   S700_BT_CODE_2101.TEST_TEMP[3] := B#16#0;
   S700_BT_CODE_2101.TEST_TEMP[4] := B#16#0;
   S700_BT_CODE_2101.TEST_TEMP[5] := B#16#0;
   S700_BT_CODE_2101.TEST_TEMP[6] := B#16#0;
   S700_BT_CODE_2101.TEST_TEMP[7] := B#16#0;
   S700_BT_CODE_2101.TEST_TEMP[8] := B#16#0;
   S700_BT_CODE_2101.TEST_TEMP[9] := B#16#0;
   S700_BT_CODE_2101.TEST_TEMP[10] := B#16#0;
   S700_BT_CODE_2101.TEST_TEMP[11] := B#16#0;
   S700_BT_CODE_2101.TEST_TEMP[12] := B#16#0;
   S700_BT_CODE_2101.TEST_TEMP[13] := B#16#0;
   S700_BT_CODE_2101.TEST_TEMP[14] := B#16#0;
   S700_BT_CODE_2101.TEST_TEMP[15] := B#16#0;
   S700_BT_CODE_2101.TEST_TEMP[16] := B#16#0;
   S700_BT_CODE_2101.TEST_TEMP[17] := B#16#0;
   S700_BT_CODE_2101.TEST_TEMP[18] := B#16#0;
   S700_BT_CODE_2101.TEST_TEMP[19] := B#16#0;
   S700_BT_CODE_2101.TEST_TEMP[20] := B#16#0;
   S700_BT_CODE_2101.TEST_TEMP[21] := B#16#0;
   S700_BT_CODE_2101.TEST_TEMP[22] := B#16#0;
   S700_BT_CODE_2101.TEST_TEMP[23] := B#16#0;
   S700_BT_CODE_2101.TEST_TEMP[24] := B#16#0;
   S700_BT_CODE_2101.TEST_TEMP[25] := B#16#0;
   S700_BT_CODE_2101.TEST_TEMP[26] := B#16#0;
   S700_BT_CODE_2101.TEST_TEMP[27] := B#16#0;
   S700_BT_CODE_2101.TEST_TEMP[28] := B#16#0;
   S700_BT_CODE_2101.TEST_TEMP[29] := B#16#0;
   S700_BT_CODE_2101.TEST_TEMP[30] := B#16#0;
   S700_BT_CODE_2101.TEST_TEMP[31] := B#16#0;
   S700_BT_CODE_2101.TEST_TEMP[32] := B#16#0;
   S700_BT_CODE_2101.TEST_TEMP[33] := B#16#0;
   S700_BT_CODE_2101.TEST_TEMP[34] := B#16#0;
   S700_BT_CODE_2101.TEST_TEMP[35] := B#16#0;
   S700_BT_CODE_2101.TEST_TEMP[36] := B#16#0;
   S700_BT_CODE_2101.TEST_TEMP[37] := B#16#0;
   S700_BT_CODE_2101.TEST_TEMP[38] := B#16#0;
   S700_BT_CODE_2101.TEST_TEMP[39] := B#16#0;
   S700_BT_CODE_2101.TEST_TEMP[40] := B#16#0;
   S700_BT_CODE_2102.STATION_MAIN := W#16#0;
   S700_BT_CODE_2102.DISTINCTION_LH_RH := W#16#0;
   S700_BT_CODE_2102.STAION_NUMBER := W#16#0;
   S700_BT_CODE_2102.BODY_TYPE_1ST := W#16#0;
   S700_BT_CODE_2102.BODY_TYPE_OPTION := W#16#0;
   S700_BT_CODE_2102.RBT1_STANDARD_WELD_DATA := W#16#0;
   S700_BT_CODE_2102.RBT2_STANDARD_WELD_DATA := W#16#0;
   S700_BT_CODE_2102.RBT3_STANDARD_WELD_DATA := W#16#0;
   S700_BT_CODE_2102.RBT4_STANDARD_WELD_DATA := W#16#0;
   S700_BT_CODE_2102.RBT5_STANDARD_WELD_DATA := W#16#0;
   S700_BT_CODE_2102.RBT6_STANDARD_WELD_DATA := W#16#0;
   S700_BT_CODE_2102.RBT7_STANDARD_WELD_DATA := W#16#0;
   S700_BT_CODE_2102.RBT8_STANDARD_WELD_DATA := W#16#0;
   S700_BT_CODE_2102.RBT9_STANDARD_WELD_DATA := W#16#0;
   S700_BT_CODE_2102.RBT10_STANDARD_WELD_DATA := W#16#0;
   S700_BT_CODE_2102.RBT11_STANDARD_WELD_DATA := W#16#0;
   S700_BT_CODE_2102.RBT12_STANDARD_WELD_DATA := W#16#0;
   S700_BT_CODE_2102.RBT13_STANDARD_WELD_DATA := W#16#0;
   S700_BT_CODE_2102.RBT14_STANDARD_WELD_DATA := W#16#0;
   S700_BT_CODE_2102.RBT15_STANDARD_WELD_DATA := W#16#0;
   S700_BT_CODE_2102.RBT16_STANDARD_WELD_DATA := W#16#0;
   S700_BT_CODE_2102.RBT17_STANDARD_WELD_DATA := W#16#0;
   S700_BT_CODE_2102.RBT18_STANDARD_WELD_DATA := W#16#0;
   S700_BT_CODE_2102.RBT19_STANDARD_WELD_DATA := W#16#0;
   S700_BT_CODE_2102.RBT20_STANDARD_WELD_DATA := W#16#0;
   S700_BT_CODE_2102.RBT21_STANDARD_WELD_DATA := W#16#0;
   S700_BT_CODE_2102.RBT22_STANDARD_WELD_DATA := W#16#0;
   S700_BT_CODE_2102.RBT23_STANDARD_WELD_DAT := W#16#0;
   S700_BT_CODE_2102.RBT24_STANDARD_WELD_DAT := W#16#0;
   S700_BT_CODE_2102.CHK_WORD := W#16#0;
   S700_BT_CODE_2102.TEST_TEMP[1] := B#16#0;
   S700_BT_CODE_2102.TEST_TEMP[2] := B#16#0;
   S700_BT_CODE_2102.TEST_TEMP[3] := B#16#0;
   S700_BT_CODE_2102.TEST_TEMP[4] := B#16#0;
   S700_BT_CODE_2102.TEST_TEMP[5] := B#16#0;
   S700_BT_CODE_2102.TEST_TEMP[6] := B#16#0;
   S700_BT_CODE_2102.TEST_TEMP[7] := B#16#0;
   S700_BT_CODE_2102.TEST_TEMP[8] := B#16#0;
   S700_BT_CODE_2102.TEST_TEMP[9] := B#16#0;
   S700_BT_CODE_2102.TEST_TEMP[10] := B#16#0;
   S700_BT_CODE_2102.TEST_TEMP[11] := B#16#0;
   S700_BT_CODE_2102.TEST_TEMP[12] := B#16#0;
   S700_BT_CODE_2102.TEST_TEMP[13] := B#16#0;
   S700_BT_CODE_2102.TEST_TEMP[14] := B#16#0;
   S700_BT_CODE_2102.TEST_TEMP[15] := B#16#0;
   S700_BT_CODE_2102.TEST_TEMP[16] := B#16#0;
   S700_BT_CODE_2102.TEST_TEMP[17] := B#16#0;
   S700_BT_CODE_2102.TEST_TEMP[18] := B#16#0;
   S700_BT_CODE_2102.TEST_TEMP[19] := B#16#0;
   S700_BT_CODE_2102.TEST_TEMP[20] := B#16#0;
   S700_BT_CODE_2102.TEST_TEMP[21] := B#16#0;
   S700_BT_CODE_2102.TEST_TEMP[22] := B#16#0;
   S700_BT_CODE_2102.TEST_TEMP[23] := B#16#0;
   S700_BT_CODE_2102.TEST_TEMP[24] := B#16#0;
   S700_BT_CODE_2102.TEST_TEMP[25] := B#16#0;
   S700_BT_CODE_2102.TEST_TEMP[26] := B#16#0;
   S700_BT_CODE_2102.TEST_TEMP[27] := B#16#0;
   S700_BT_CODE_2102.TEST_TEMP[28] := B#16#0;
   S700_BT_CODE_2102.TEST_TEMP[29] := B#16#0;
   S700_BT_CODE_2102.TEST_TEMP[30] := B#16#0;
   S700_BT_CODE_2102.TEST_TEMP[31] := B#16#0;
   S700_BT_CODE_2102.TEST_TEMP[32] := B#16#0;
   S700_BT_CODE_2102.TEST_TEMP[33] := B#16#0;
   S700_BT_CODE_2102.TEST_TEMP[34] := B#16#0;
   S700_BT_CODE_2102.TEST_TEMP[35] := B#16#0;
   S700_BT_CODE_2102.TEST_TEMP[36] := B#16#0;
   S700_BT_CODE_2102.TEST_TEMP[37] := B#16#0;
   S700_BT_CODE_2102.TEST_TEMP[38] := B#16#0;
   S700_BT_CODE_2102.TEST_TEMP[39] := B#16#0;
   S700_BT_CODE_2102.TEST_TEMP[40] := B#16#0;
   S700_BT_CODE_2103.STATION_MAIN := W#16#0;
   S700_BT_CODE_2103.DISTINCTION_LH_RH := W#16#0;
   S700_BT_CODE_2103.STAION_NUMBER := W#16#0;
   S700_BT_CODE_2103.BODY_TYPE_1ST := W#16#0;
   S700_BT_CODE_2103.BODY_TYPE_OPTION := W#16#0;
   S700_BT_CODE_2103.RBT1_STANDARD_WELD_DATA := W#16#0;
   S700_BT_CODE_2103.RBT2_STANDARD_WELD_DATA := W#16#0;
   S700_BT_CODE_2103.RBT3_STANDARD_WELD_DATA := W#16#0;
   S700_BT_CODE_2103.RBT4_STANDARD_WELD_DATA := W#16#0;
   S700_BT_CODE_2103.RBT5_STANDARD_WELD_DATA := W#16#0;
   S700_BT_CODE_2103.RBT6_STANDARD_WELD_DATA := W#16#0;
   S700_BT_CODE_2103.RBT7_STANDARD_WELD_DATA := W#16#0;
   S700_BT_CODE_2103.RBT8_STANDARD_WELD_DATA := W#16#0;
   S700_BT_CODE_2103.RBT9_STANDARD_WELD_DATA := W#16#0;
   S700_BT_CODE_2103.RBT10_STANDARD_WELD_DATA := W#16#0;
   S700_BT_CODE_2103.RBT11_STANDARD_WELD_DATA := W#16#0;
   S700_BT_CODE_2103.RBT12_STANDARD_WELD_DATA := W#16#0;
   S700_BT_CODE_2103.RBT13_STANDARD_WELD_DATA := W#16#0;
   S700_BT_CODE_2103.RBT14_STANDARD_WELD_DATA := W#16#0;
   S700_BT_CODE_2103.RBT15_STANDARD_WELD_DATA := W#16#0;
   S700_BT_CODE_2103.RBT16_STANDARD_WELD_DATA := W#16#0;
   S700_BT_CODE_2103.RBT17_STANDARD_WELD_DATA := W#16#0;
   S700_BT_CODE_2103.RBT18_STANDARD_WELD_DATA := W#16#0;
   S700_BT_CODE_2103.RBT19_STANDARD_WELD_DATA := W#16#0;
   S700_BT_CODE_2103.RBT20_STANDARD_WELD_DATA := W#16#0;
   S700_BT_CODE_2103.RBT21_STANDARD_WELD_DATA := W#16#0;
   S700_BT_CODE_2103.RBT22_STANDARD_WELD_DATA := W#16#0;
   S700_BT_CODE_2103.RBT23_STANDARD_WELD_DAT := W#16#0;
   S700_BT_CODE_2103.RBT24_STANDARD_WELD_DAT := W#16#0;
   S700_BT_CODE_2103.CHK_WORD := W#16#0;
   S700_BT_CODE_2103.TEST_TEMP[1] := B#16#0;
   S700_BT_CODE_2103.TEST_TEMP[2] := B#16#0;
   S700_BT_CODE_2103.TEST_TEMP[3] := B#16#0;
   S700_BT_CODE_2103.TEST_TEMP[4] := B#16#0;
   S700_BT_CODE_2103.TEST_TEMP[5] := B#16#0;
   S700_BT_CODE_2103.TEST_TEMP[6] := B#16#0;
   S700_BT_CODE_2103.TEST_TEMP[7] := B#16#0;
   S700_BT_CODE_2103.TEST_TEMP[8] := B#16#0;
   S700_BT_CODE_2103.TEST_TEMP[9] := B#16#0;
   S700_BT_CODE_2103.TEST_TEMP[10] := B#16#0;
   S700_BT_CODE_2103.TEST_TEMP[11] := B#16#0;
   S700_BT_CODE_2103.TEST_TEMP[12] := B#16#0;
   S700_BT_CODE_2103.TEST_TEMP[13] := B#16#0;
   S700_BT_CODE_2103.TEST_TEMP[14] := B#16#0;
   S700_BT_CODE_2103.TEST_TEMP[15] := B#16#0;
   S700_BT_CODE_2103.TEST_TEMP[16] := B#16#0;
   S700_BT_CODE_2103.TEST_TEMP[17] := B#16#0;
   S700_BT_CODE_2103.TEST_TEMP[18] := B#16#0;
   S700_BT_CODE_2103.TEST_TEMP[19] := B#16#0;
   S700_BT_CODE_2103.TEST_TEMP[20] := B#16#0;
   S700_BT_CODE_2103.TEST_TEMP[21] := B#16#0;
   S700_BT_CODE_2103.TEST_TEMP[22] := B#16#0;
   S700_BT_CODE_2103.TEST_TEMP[23] := B#16#0;
   S700_BT_CODE_2103.TEST_TEMP[24] := B#16#0;
   S700_BT_CODE_2103.TEST_TEMP[25] := B#16#0;
   S700_BT_CODE_2103.TEST_TEMP[26] := B#16#0;
   S700_BT_CODE_2103.TEST_TEMP[27] := B#16#0;
   S700_BT_CODE_2103.TEST_TEMP[28] := B#16#0;
   S700_BT_CODE_2103.TEST_TEMP[29] := B#16#0;
   S700_BT_CODE_2103.TEST_TEMP[30] := B#16#0;
   S700_BT_CODE_2103.TEST_TEMP[31] := B#16#0;
   S700_BT_CODE_2103.TEST_TEMP[32] := B#16#0;
   S700_BT_CODE_2103.TEST_TEMP[33] := B#16#0;
   S700_BT_CODE_2103.TEST_TEMP[34] := B#16#0;
   S700_BT_CODE_2103.TEST_TEMP[35] := B#16#0;
   S700_BT_CODE_2103.TEST_TEMP[36] := B#16#0;
   S700_BT_CODE_2103.TEST_TEMP[37] := B#16#0;
   S700_BT_CODE_2103.TEST_TEMP[38] := B#16#0;
   S700_BT_CODE_2103.TEST_TEMP[39] := B#16#0;
   S700_BT_CODE_2103.TEST_TEMP[40] := B#16#0;
   S700_BT_CODE_2104.STATION_MAIN := W#16#0;
   S700_BT_CODE_2104.DISTINCTION_LH_RH := W#16#0;
   S700_BT_CODE_2104.STAION_NUMBER := W#16#0;
   S700_BT_CODE_2104.BODY_TYPE_1ST := W#16#0;
   S700_BT_CODE_2104.BODY_TYPE_OPTION := W#16#0;
   S700_BT_CODE_2104.RBT1_STANDARD_WELD_DATA := W#16#0;
   S700_BT_CODE_2104.RBT2_STANDARD_WELD_DATA := W#16#0;
   S700_BT_CODE_2104.RBT3_STANDARD_WELD_DATA := W#16#0;
   S700_BT_CODE_2104.RBT4_STANDARD_WELD_DATA := W#16#0;
   S700_BT_CODE_2104.RBT5_STANDARD_WELD_DATA := W#16#0;
   S700_BT_CODE_2104.RBT6_STANDARD_WELD_DATA := W#16#0;
   S700_BT_CODE_2104.RBT7_STANDARD_WELD_DATA := W#16#0;
   S700_BT_CODE_2104.RBT8_STANDARD_WELD_DATA := W#16#0;
   S700_BT_CODE_2104.RBT9_STANDARD_WELD_DATA := W#16#0;
   S700_BT_CODE_2104.RBT10_STANDARD_WELD_DATA := W#16#0;
   S700_BT_CODE_2104.RBT11_STANDARD_WELD_DATA := W#16#0;
   S700_BT_CODE_2104.RBT12_STANDARD_WELD_DATA := W#16#0;
   S700_BT_CODE_2104.RBT13_STANDARD_WELD_DATA := W#16#0;
   S700_BT_CODE_2104.RBT14_STANDARD_WELD_DATA := W#16#0;
   S700_BT_CODE_2104.RBT15_STANDARD_WELD_DATA := W#16#0;
   S700_BT_CODE_2104.RBT16_STANDARD_WELD_DATA := W#16#0;
   S700_BT_CODE_2104.RBT17_STANDARD_WELD_DATA := W#16#0;
   S700_BT_CODE_2104.RBT18_STANDARD_WELD_DATA := W#16#0;
   S700_BT_CODE_2104.RBT19_STANDARD_WELD_DATA := W#16#0;
   S700_BT_CODE_2104.RBT20_STANDARD_WELD_DATA := W#16#0;
   S700_BT_CODE_2104.RBT21_STANDARD_WELD_DATA := W#16#0;
   S700_BT_CODE_2104.RBT22_STANDARD_WELD_DATA := W#16#0;
   S700_BT_CODE_2104.RBT23_STANDARD_WELD_DAT := W#16#0;
   S700_BT_CODE_2104.RBT24_STANDARD_WELD_DAT := W#16#0;
   S700_BT_CODE_2104.CHK_WORD := W#16#0;
   S700_BT_CODE_2104.TEST_TEMP[1] := B#16#0;
   S700_BT_CODE_2104.TEST_TEMP[2] := B#16#0;
   S700_BT_CODE_2104.TEST_TEMP[3] := B#16#0;
   S700_BT_CODE_2104.TEST_TEMP[4] := B#16#0;
   S700_BT_CODE_2104.TEST_TEMP[5] := B#16#0;
   S700_BT_CODE_2104.TEST_TEMP[6] := B#16#0;
   S700_BT_CODE_2104.TEST_TEMP[7] := B#16#0;
   S700_BT_CODE_2104.TEST_TEMP[8] := B#16#0;
   S700_BT_CODE_2104.TEST_TEMP[9] := B#16#0;
   S700_BT_CODE_2104.TEST_TEMP[10] := B#16#0;
   S700_BT_CODE_2104.TEST_TEMP[11] := B#16#0;
   S700_BT_CODE_2104.TEST_TEMP[12] := B#16#0;
   S700_BT_CODE_2104.TEST_TEMP[13] := B#16#0;
   S700_BT_CODE_2104.TEST_TEMP[14] := B#16#0;
   S700_BT_CODE_2104.TEST_TEMP[15] := B#16#0;
   S700_BT_CODE_2104.TEST_TEMP[16] := B#16#0;
   S700_BT_CODE_2104.TEST_TEMP[17] := B#16#0;
   S700_BT_CODE_2104.TEST_TEMP[18] := B#16#0;
   S700_BT_CODE_2104.TEST_TEMP[19] := B#16#0;
   S700_BT_CODE_2104.TEST_TEMP[20] := B#16#0;
   S700_BT_CODE_2104.TEST_TEMP[21] := B#16#0;
   S700_BT_CODE_2104.TEST_TEMP[22] := B#16#0;
   S700_BT_CODE_2104.TEST_TEMP[23] := B#16#0;
   S700_BT_CODE_2104.TEST_TEMP[24] := B#16#0;
   S700_BT_CODE_2104.TEST_TEMP[25] := B#16#0;
   S700_BT_CODE_2104.TEST_TEMP[26] := B#16#0;
   S700_BT_CODE_2104.TEST_TEMP[27] := B#16#0;
   S700_BT_CODE_2104.TEST_TEMP[28] := B#16#0;
   S700_BT_CODE_2104.TEST_TEMP[29] := B#16#0;
   S700_BT_CODE_2104.TEST_TEMP[30] := B#16#0;
   S700_BT_CODE_2104.TEST_TEMP[31] := B#16#0;
   S700_BT_CODE_2104.TEST_TEMP[32] := B#16#0;
   S700_BT_CODE_2104.TEST_TEMP[33] := B#16#0;
   S700_BT_CODE_2104.TEST_TEMP[34] := B#16#0;
   S700_BT_CODE_2104.TEST_TEMP[35] := B#16#0;
   S700_BT_CODE_2104.TEST_TEMP[36] := B#16#0;
   S700_BT_CODE_2104.TEST_TEMP[37] := B#16#0;
   S700_BT_CODE_2104.TEST_TEMP[38] := B#16#0;
   S700_BT_CODE_2104.TEST_TEMP[39] := B#16#0;
   S700_BT_CODE_2104.TEST_TEMP[40] := B#16#0;
   S700_BT_CODE_2105.STATION_MAIN := W#16#0;
   S700_BT_CODE_2105.DISTINCTION_LH_RH := W#16#0;
   S700_BT_CODE_2105.STAION_NUMBER := W#16#0;
   S700_BT_CODE_2105.BODY_TYPE_1ST := W#16#0;
   S700_BT_CODE_2105.BODY_TYPE_OPTION := W#16#0;
   S700_BT_CODE_2105.RBT1_STANDARD_WELD_DATA := W#16#0;
   S700_BT_CODE_2105.RBT2_STANDARD_WELD_DATA := W#16#0;
   S700_BT_CODE_2105.RBT3_STANDARD_WELD_DATA := W#16#0;
   S700_BT_CODE_2105.RBT4_STANDARD_WELD_DATA := W#16#0;
   S700_BT_CODE_2105.RBT5_STANDARD_WELD_DATA := W#16#0;
   S700_BT_CODE_2105.RBT6_STANDARD_WELD_DATA := W#16#0;
   S700_BT_CODE_2105.RBT7_STANDARD_WELD_DATA := W#16#0;
   S700_BT_CODE_2105.RBT8_STANDARD_WELD_DATA := W#16#0;
   S700_BT_CODE_2105.RBT9_STANDARD_WELD_DATA := W#16#0;
   S700_BT_CODE_2105.RBT10_STANDARD_WELD_DATA := W#16#0;
   S700_BT_CODE_2105.RBT11_STANDARD_WELD_DATA := W#16#0;
   S700_BT_CODE_2105.RBT12_STANDARD_WELD_DATA := W#16#0;
   S700_BT_CODE_2105.RBT13_STANDARD_WELD_DATA := W#16#0;
   S700_BT_CODE_2105.RBT14_STANDARD_WELD_DATA := W#16#0;
   S700_BT_CODE_2105.RBT15_STANDARD_WELD_DATA := W#16#0;
   S700_BT_CODE_2105.RBT16_STANDARD_WELD_DATA := W#16#0;
   S700_BT_CODE_2105.RBT17_STANDARD_WELD_DATA := W#16#0;
   S700_BT_CODE_2105.RBT18_STANDARD_WELD_DATA := W#16#0;
   S700_BT_CODE_2105.RBT19_STANDARD_WELD_DATA := W#16#0;
   S700_BT_CODE_2105.RBT20_STANDARD_WELD_DATA := W#16#0;
   S700_BT_CODE_2105.RBT21_STANDARD_WELD_DATA := W#16#0;
   S700_BT_CODE_2105.RBT22_STANDARD_WELD_DATA := W#16#0;
   S700_BT_CODE_2105.RBT23_STANDARD_WELD_DAT := W#16#0;
   S700_BT_CODE_2105.RBT24_STANDARD_WELD_DAT := W#16#0;
   S700_BT_CODE_2105.CHK_WORD := W#16#0;
   S700_BT_CODE_2105.TEST_TEMP[1] := B#16#0;
   S700_BT_CODE_2105.TEST_TEMP[2] := B#16#0;
   S700_BT_CODE_2105.TEST_TEMP[3] := B#16#0;
   S700_BT_CODE_2105.TEST_TEMP[4] := B#16#0;
   S700_BT_CODE_2105.TEST_TEMP[5] := B#16#0;
   S700_BT_CODE_2105.TEST_TEMP[6] := B#16#0;
   S700_BT_CODE_2105.TEST_TEMP[7] := B#16#0;
   S700_BT_CODE_2105.TEST_TEMP[8] := B#16#0;
   S700_BT_CODE_2105.TEST_TEMP[9] := B#16#0;
   S700_BT_CODE_2105.TEST_TEMP[10] := B#16#0;
   S700_BT_CODE_2105.TEST_TEMP[11] := B#16#0;
   S700_BT_CODE_2105.TEST_TEMP[12] := B#16#0;
   S700_BT_CODE_2105.TEST_TEMP[13] := B#16#0;
   S700_BT_CODE_2105.TEST_TEMP[14] := B#16#0;
   S700_BT_CODE_2105.TEST_TEMP[15] := B#16#0;
   S700_BT_CODE_2105.TEST_TEMP[16] := B#16#0;
   S700_BT_CODE_2105.TEST_TEMP[17] := B#16#0;
   S700_BT_CODE_2105.TEST_TEMP[18] := B#16#0;
   S700_BT_CODE_2105.TEST_TEMP[19] := B#16#0;
   S700_BT_CODE_2105.TEST_TEMP[20] := B#16#0;
   S700_BT_CODE_2105.TEST_TEMP[21] := B#16#0;
   S700_BT_CODE_2105.TEST_TEMP[22] := B#16#0;
   S700_BT_CODE_2105.TEST_TEMP[23] := B#16#0;
   S700_BT_CODE_2105.TEST_TEMP[24] := B#16#0;
   S700_BT_CODE_2105.TEST_TEMP[25] := B#16#0;
   S700_BT_CODE_2105.TEST_TEMP[26] := B#16#0;
   S700_BT_CODE_2105.TEST_TEMP[27] := B#16#0;
   S700_BT_CODE_2105.TEST_TEMP[28] := B#16#0;
   S700_BT_CODE_2105.TEST_TEMP[29] := B#16#0;
   S700_BT_CODE_2105.TEST_TEMP[30] := B#16#0;
   S700_BT_CODE_2105.TEST_TEMP[31] := B#16#0;
   S700_BT_CODE_2105.TEST_TEMP[32] := B#16#0;
   S700_BT_CODE_2105.TEST_TEMP[33] := B#16#0;
   S700_BT_CODE_2105.TEST_TEMP[34] := B#16#0;
   S700_BT_CODE_2105.TEST_TEMP[35] := B#16#0;
   S700_BT_CODE_2105.TEST_TEMP[36] := B#16#0;
   S700_BT_CODE_2105.TEST_TEMP[37] := B#16#0;
   S700_BT_CODE_2105.TEST_TEMP[38] := B#16#0;
   S700_BT_CODE_2105.TEST_TEMP[39] := B#16#0;
   S700_BT_CODE_2105.TEST_TEMP[40] := B#16#0;
   S700_BT_CODE_2106.STATION_MAIN := W#16#0;
   S700_BT_CODE_2106.DISTINCTION_LH_RH := W#16#0;
   S700_BT_CODE_2106.STAION_NUMBER := W#16#0;
   S700_BT_CODE_2106.BODY_TYPE_1ST := W#16#0;
   S700_BT_CODE_2106.BODY_TYPE_OPTION := W#16#0;
   S700_BT_CODE_2106.RBT1_STANDARD_WELD_DATA := W#16#0;
   S700_BT_CODE_2106.RBT2_STANDARD_WELD_DATA := W#16#0;
   S700_BT_CODE_2106.RBT3_STANDARD_WELD_DATA := W#16#0;
   S700_BT_CODE_2106.RBT4_STANDARD_WELD_DATA := W#16#0;
   S700_BT_CODE_2106.RBT5_STANDARD_WELD_DATA := W#16#0;
   S700_BT_CODE_2106.RBT6_STANDARD_WELD_DATA := W#16#0;
   S700_BT_CODE_2106.RBT7_STANDARD_WELD_DATA := W#16#0;
   S700_BT_CODE_2106.RBT8_STANDARD_WELD_DATA := W#16#0;
   S700_BT_CODE_2106.RBT9_STANDARD_WELD_DATA := W#16#0;
   S700_BT_CODE_2106.RBT10_STANDARD_WELD_DATA := W#16#0;
   S700_BT_CODE_2106.RBT11_STANDARD_WELD_DATA := W#16#0;
   S700_BT_CODE_2106.RBT12_STANDARD_WELD_DATA := W#16#0;
   S700_BT_CODE_2106.RBT13_STANDARD_WELD_DATA := W#16#0;
   S700_BT_CODE_2106.RBT14_STANDARD_WELD_DATA := W#16#0;
   S700_BT_CODE_2106.RBT15_STANDARD_WELD_DATA := W#16#0;
   S700_BT_CODE_2106.RBT16_STANDARD_WELD_DATA := W#16#0;
   S700_BT_CODE_2106.RBT17_STANDARD_WELD_DATA := W#16#0;
   S700_BT_CODE_2106.RBT18_STANDARD_WELD_DATA := W#16#0;
   S700_BT_CODE_2106.RBT19_STANDARD_WELD_DATA := W#16#0;
   S700_BT_CODE_2106.RBT20_STANDARD_WELD_DATA := W#16#0;
   S700_BT_CODE_2106.RBT21_STANDARD_WELD_DATA := W#16#0;
   S700_BT_CODE_2106.RBT22_STANDARD_WELD_DATA := W#16#0;
   S700_BT_CODE_2106.RBT23_STANDARD_WELD_DAT := W#16#0;
   S700_BT_CODE_2106.RBT24_STANDARD_WELD_DAT := W#16#0;
   S700_BT_CODE_2106.CHK_WORD := W#16#0;
   S700_BT_CODE_2106.TEST_TEMP[1] := B#16#0;
   S700_BT_CODE_2106.TEST_TEMP[2] := B#16#0;
   S700_BT_CODE_2106.TEST_TEMP[3] := B#16#0;
   S700_BT_CODE_2106.TEST_TEMP[4] := B#16#0;
   S700_BT_CODE_2106.TEST_TEMP[5] := B#16#0;
   S700_BT_CODE_2106.TEST_TEMP[6] := B#16#0;
   S700_BT_CODE_2106.TEST_TEMP[7] := B#16#0;
   S700_BT_CODE_2106.TEST_TEMP[8] := B#16#0;
   S700_BT_CODE_2106.TEST_TEMP[9] := B#16#0;
   S700_BT_CODE_2106.TEST_TEMP[10] := B#16#0;
   S700_BT_CODE_2106.TEST_TEMP[11] := B#16#0;
   S700_BT_CODE_2106.TEST_TEMP[12] := B#16#0;
   S700_BT_CODE_2106.TEST_TEMP[13] := B#16#0;
   S700_BT_CODE_2106.TEST_TEMP[14] := B#16#0;
   S700_BT_CODE_2106.TEST_TEMP[15] := B#16#0;
   S700_BT_CODE_2106.TEST_TEMP[16] := B#16#0;
   S700_BT_CODE_2106.TEST_TEMP[17] := B#16#0;
   S700_BT_CODE_2106.TEST_TEMP[18] := B#16#0;
   S700_BT_CODE_2106.TEST_TEMP[19] := B#16#0;
   S700_BT_CODE_2106.TEST_TEMP[20] := B#16#0;
   S700_BT_CODE_2106.TEST_TEMP[21] := B#16#0;
   S700_BT_CODE_2106.TEST_TEMP[22] := B#16#0;
   S700_BT_CODE_2106.TEST_TEMP[23] := B#16#0;
   S700_BT_CODE_2106.TEST_TEMP[24] := B#16#0;
   S700_BT_CODE_2106.TEST_TEMP[25] := B#16#0;
   S700_BT_CODE_2106.TEST_TEMP[26] := B#16#0;
   S700_BT_CODE_2106.TEST_TEMP[27] := B#16#0;
   S700_BT_CODE_2106.TEST_TEMP[28] := B#16#0;
   S700_BT_CODE_2106.TEST_TEMP[29] := B#16#0;
   S700_BT_CODE_2106.TEST_TEMP[30] := B#16#0;
   S700_BT_CODE_2106.TEST_TEMP[31] := B#16#0;
   S700_BT_CODE_2106.TEST_TEMP[32] := B#16#0;
   S700_BT_CODE_2106.TEST_TEMP[33] := B#16#0;
   S700_BT_CODE_2106.TEST_TEMP[34] := B#16#0;
   S700_BT_CODE_2106.TEST_TEMP[35] := B#16#0;
   S700_BT_CODE_2106.TEST_TEMP[36] := B#16#0;
   S700_BT_CODE_2106.TEST_TEMP[37] := B#16#0;
   S700_BT_CODE_2106.TEST_TEMP[38] := B#16#0;
   S700_BT_CODE_2106.TEST_TEMP[39] := B#16#0;
   S700_BT_CODE_2106.TEST_TEMP[40] := B#16#0;
   S700_BT_CODE_2107.STATION_MAIN := W#16#0;
   S700_BT_CODE_2107.DISTINCTION_LH_RH := W#16#0;
   S700_BT_CODE_2107.STAION_NUMBER := W#16#0;
   S700_BT_CODE_2107.BODY_TYPE_1ST := W#16#0;
   S700_BT_CODE_2107.BODY_TYPE_OPTION := W#16#0;
   S700_BT_CODE_2107.RBT1_STANDARD_WELD_DATA := W#16#0;
   S700_BT_CODE_2107.RBT2_STANDARD_WELD_DATA := W#16#0;
   S700_BT_CODE_2107.RBT3_STANDARD_WELD_DATA := W#16#0;
   S700_BT_CODE_2107.RBT4_STANDARD_WELD_DATA := W#16#0;
   S700_BT_CODE_2107.RBT5_STANDARD_WELD_DATA := W#16#0;
   S700_BT_CODE_2107.RBT6_STANDARD_WELD_DATA := W#16#0;
   S700_BT_CODE_2107.RBT7_STANDARD_WELD_DATA := W#16#0;
   S700_BT_CODE_2107.RBT8_STANDARD_WELD_DATA := W#16#0;
   S700_BT_CODE_2107.RBT9_STANDARD_WELD_DATA := W#16#0;
   S700_BT_CODE_2107.RBT10_STANDARD_WELD_DATA := W#16#0;
   S700_BT_CODE_2107.RBT11_STANDARD_WELD_DATA := W#16#0;
   S700_BT_CODE_2107.RBT12_STANDARD_WELD_DATA := W#16#0;
   S700_BT_CODE_2107.RBT13_STANDARD_WELD_DATA := W#16#0;
   S700_BT_CODE_2107.RBT14_STANDARD_WELD_DATA := W#16#0;
   S700_BT_CODE_2107.RBT15_STANDARD_WELD_DATA := W#16#0;
   S700_BT_CODE_2107.RBT16_STANDARD_WELD_DATA := W#16#0;
   S700_BT_CODE_2107.RBT17_STANDARD_WELD_DATA := W#16#0;
   S700_BT_CODE_2107.RBT18_STANDARD_WELD_DATA := W#16#0;
   S700_BT_CODE_2107.RBT19_STANDARD_WELD_DATA := W#16#0;
   S700_BT_CODE_2107.RBT20_STANDARD_WELD_DATA := W#16#0;
   S700_BT_CODE_2107.RBT21_STANDARD_WELD_DATA := W#16#0;
   S700_BT_CODE_2107.RBT22_STANDARD_WELD_DATA := W#16#0;
   S700_BT_CODE_2107.RBT23_STANDARD_WELD_DAT := W#16#0;
   S700_BT_CODE_2107.RBT24_STANDARD_WELD_DAT := W#16#0;
   S700_BT_CODE_2107.CHK_WORD := W#16#0;
   S700_BT_CODE_2107.TEST_TEMP[1] := B#16#0;
   S700_BT_CODE_2107.TEST_TEMP[2] := B#16#0;
   S700_BT_CODE_2107.TEST_TEMP[3] := B#16#0;
   S700_BT_CODE_2107.TEST_TEMP[4] := B#16#0;
   S700_BT_CODE_2107.TEST_TEMP[5] := B#16#0;
   S700_BT_CODE_2107.TEST_TEMP[6] := B#16#0;
   S700_BT_CODE_2107.TEST_TEMP[7] := B#16#0;
   S700_BT_CODE_2107.TEST_TEMP[8] := B#16#0;
   S700_BT_CODE_2107.TEST_TEMP[9] := B#16#0;
   S700_BT_CODE_2107.TEST_TEMP[10] := B#16#0;
   S700_BT_CODE_2107.TEST_TEMP[11] := B#16#0;
   S700_BT_CODE_2107.TEST_TEMP[12] := B#16#0;
   S700_BT_CODE_2107.TEST_TEMP[13] := B#16#0;
   S700_BT_CODE_2107.TEST_TEMP[14] := B#16#0;
   S700_BT_CODE_2107.TEST_TEMP[15] := B#16#0;
   S700_BT_CODE_2107.TEST_TEMP[16] := B#16#0;
   S700_BT_CODE_2107.TEST_TEMP[17] := B#16#0;
   S700_BT_CODE_2107.TEST_TEMP[18] := B#16#0;
   S700_BT_CODE_2107.TEST_TEMP[19] := B#16#0;
   S700_BT_CODE_2107.TEST_TEMP[20] := B#16#0;
   S700_BT_CODE_2107.TEST_TEMP[21] := B#16#0;
   S700_BT_CODE_2107.TEST_TEMP[22] := B#16#0;
   S700_BT_CODE_2107.TEST_TEMP[23] := B#16#0;
   S700_BT_CODE_2107.TEST_TEMP[24] := B#16#0;
   S700_BT_CODE_2107.TEST_TEMP[25] := B#16#0;
   S700_BT_CODE_2107.TEST_TEMP[26] := B#16#0;
   S700_BT_CODE_2107.TEST_TEMP[27] := B#16#0;
   S700_BT_CODE_2107.TEST_TEMP[28] := B#16#0;
   S700_BT_CODE_2107.TEST_TEMP[29] := B#16#0;
   S700_BT_CODE_2107.TEST_TEMP[30] := B#16#0;
   S700_BT_CODE_2107.TEST_TEMP[31] := B#16#0;
   S700_BT_CODE_2107.TEST_TEMP[32] := B#16#0;
   S700_BT_CODE_2107.TEST_TEMP[33] := B#16#0;
   S700_BT_CODE_2107.TEST_TEMP[34] := B#16#0;
   S700_BT_CODE_2107.TEST_TEMP[35] := B#16#0;
   S700_BT_CODE_2107.TEST_TEMP[36] := B#16#0;
   S700_BT_CODE_2107.TEST_TEMP[37] := B#16#0;
   S700_BT_CODE_2107.TEST_TEMP[38] := B#16#0;
   S700_BT_CODE_2107.TEST_TEMP[39] := B#16#0;
   S700_BT_CODE_2107.TEST_TEMP[40] := B#16#0;
   S700_BT_CODE_2108.STATION_MAIN := W#16#0;
   S700_BT_CODE_2108.DISTINCTION_LH_RH := W#16#0;
   S700_BT_CODE_2108.STAION_NUMBER := W#16#0;
   S700_BT_CODE_2108.BODY_TYPE_1ST := W#16#0;
   S700_BT_CODE_2108.BODY_TYPE_OPTION := W#16#0;
   S700_BT_CODE_2108.RBT1_STANDARD_WELD_DATA := W#16#0;
   S700_BT_CODE_2108.RBT2_STANDARD_WELD_DATA := W#16#0;
   S700_BT_CODE_2108.RBT3_STANDARD_WELD_DATA := W#16#0;
   S700_BT_CODE_2108.RBT4_STANDARD_WELD_DATA := W#16#0;
   S700_BT_CODE_2108.RBT5_STANDARD_WELD_DATA := W#16#0;
   S700_BT_CODE_2108.RBT6_STANDARD_WELD_DATA := W#16#0;
   S700_BT_CODE_2108.RBT7_STANDARD_WELD_DATA := W#16#0;
   S700_BT_CODE_2108.RBT8_STANDARD_WELD_DATA := W#16#0;
   S700_BT_CODE_2108.RBT9_STANDARD_WELD_DATA := W#16#0;
   S700_BT_CODE_2108.RBT10_STANDARD_WELD_DATA := W#16#0;
   S700_BT_CODE_2108.RBT11_STANDARD_WELD_DATA := W#16#0;
   S700_BT_CODE_2108.RBT12_STANDARD_WELD_DATA := W#16#0;
   S700_BT_CODE_2108.RBT13_STANDARD_WELD_DATA := W#16#0;
   S700_BT_CODE_2108.RBT14_STANDARD_WELD_DATA := W#16#0;
   S700_BT_CODE_2108.RBT15_STANDARD_WELD_DATA := W#16#0;
   S700_BT_CODE_2108.RBT16_STANDARD_WELD_DATA := W#16#0;
   S700_BT_CODE_2108.RBT17_STANDARD_WELD_DATA := W#16#0;
   S700_BT_CODE_2108.RBT18_STANDARD_WELD_DATA := W#16#0;
   S700_BT_CODE_2108.RBT19_STANDARD_WELD_DATA := W#16#0;
   S700_BT_CODE_2108.RBT20_STANDARD_WELD_DATA := W#16#0;
   S700_BT_CODE_2108.RBT21_STANDARD_WELD_DATA := W#16#0;
   S700_BT_CODE_2108.RBT22_STANDARD_WELD_DATA := W#16#0;
   S700_BT_CODE_2108.RBT23_STANDARD_WELD_DAT := W#16#0;
   S700_BT_CODE_2108.RBT24_STANDARD_WELD_DAT := W#16#0;
   S700_BT_CODE_2108.CHK_WORD := W#16#0;
   S700_BT_CODE_2108.TEST_TEMP[1] := B#16#0;
   S700_BT_CODE_2108.TEST_TEMP[2] := B#16#0;
   S700_BT_CODE_2108.TEST_TEMP[3] := B#16#0;
   S700_BT_CODE_2108.TEST_TEMP[4] := B#16#0;
   S700_BT_CODE_2108.TEST_TEMP[5] := B#16#0;
   S700_BT_CODE_2108.TEST_TEMP[6] := B#16#0;
   S700_BT_CODE_2108.TEST_TEMP[7] := B#16#0;
   S700_BT_CODE_2108.TEST_TEMP[8] := B#16#0;
   S700_BT_CODE_2108.TEST_TEMP[9] := B#16#0;
   S700_BT_CODE_2108.TEST_TEMP[10] := B#16#0;
   S700_BT_CODE_2108.TEST_TEMP[11] := B#16#0;
   S700_BT_CODE_2108.TEST_TEMP[12] := B#16#0;
   S700_BT_CODE_2108.TEST_TEMP[13] := B#16#0;
   S700_BT_CODE_2108.TEST_TEMP[14] := B#16#0;
   S700_BT_CODE_2108.TEST_TEMP[15] := B#16#0;
   S700_BT_CODE_2108.TEST_TEMP[16] := B#16#0;
   S700_BT_CODE_2108.TEST_TEMP[17] := B#16#0;
   S700_BT_CODE_2108.TEST_TEMP[18] := B#16#0;
   S700_BT_CODE_2108.TEST_TEMP[19] := B#16#0;
   S700_BT_CODE_2108.TEST_TEMP[20] := B#16#0;
   S700_BT_CODE_2108.TEST_TEMP[21] := B#16#0;
   S700_BT_CODE_2108.TEST_TEMP[22] := B#16#0;
   S700_BT_CODE_2108.TEST_TEMP[23] := B#16#0;
   S700_BT_CODE_2108.TEST_TEMP[24] := B#16#0;
   S700_BT_CODE_2108.TEST_TEMP[25] := B#16#0;
   S700_BT_CODE_2108.TEST_TEMP[26] := B#16#0;
   S700_BT_CODE_2108.TEST_TEMP[27] := B#16#0;
   S700_BT_CODE_2108.TEST_TEMP[28] := B#16#0;
   S700_BT_CODE_2108.TEST_TEMP[29] := B#16#0;
   S700_BT_CODE_2108.TEST_TEMP[30] := B#16#0;
   S700_BT_CODE_2108.TEST_TEMP[31] := B#16#0;
   S700_BT_CODE_2108.TEST_TEMP[32] := B#16#0;
   S700_BT_CODE_2108.TEST_TEMP[33] := B#16#0;
   S700_BT_CODE_2108.TEST_TEMP[34] := B#16#0;
   S700_BT_CODE_2108.TEST_TEMP[35] := B#16#0;
   S700_BT_CODE_2108.TEST_TEMP[36] := B#16#0;
   S700_BT_CODE_2108.TEST_TEMP[37] := B#16#0;
   S700_BT_CODE_2108.TEST_TEMP[38] := B#16#0;
   S700_BT_CODE_2108.TEST_TEMP[39] := B#16#0;
   S700_BT_CODE_2108.TEST_TEMP[40] := B#16#0;
   S700_BT_CODE_2109.STATION_MAIN := W#16#0;
   S700_BT_CODE_2109.DISTINCTION_LH_RH := W#16#0;
   S700_BT_CODE_2109.STAION_NUMBER := W#16#0;
   S700_BT_CODE_2109.BODY_TYPE_1ST := W#16#0;
   S700_BT_CODE_2109.BODY_TYPE_OPTION := W#16#0;
   S700_BT_CODE_2109.RBT1_STANDARD_WELD_DATA := W#16#0;
   S700_BT_CODE_2109.RBT2_STANDARD_WELD_DATA := W#16#0;
   S700_BT_CODE_2109.RBT3_STANDARD_WELD_DATA := W#16#0;
   S700_BT_CODE_2109.RBT4_STANDARD_WELD_DATA := W#16#0;
   S700_BT_CODE_2109.RBT5_STANDARD_WELD_DATA := W#16#0;
   S700_BT_CODE_2109.RBT6_STANDARD_WELD_DATA := W#16#0;
   S700_BT_CODE_2109.RBT7_STANDARD_WELD_DATA := W#16#0;
   S700_BT_CODE_2109.RBT8_STANDARD_WELD_DATA := W#16#0;
   S700_BT_CODE_2109.RBT9_STANDARD_WELD_DATA := W#16#0;
   S700_BT_CODE_2109.RBT10_STANDARD_WELD_DATA := W#16#0;
   S700_BT_CODE_2109.RBT11_STANDARD_WELD_DATA := W#16#0;
   S700_BT_CODE_2109.RBT12_STANDARD_WELD_DATA := W#16#0;
   S700_BT_CODE_2109.RBT13_STANDARD_WELD_DATA := W#16#0;
   S700_BT_CODE_2109.RBT14_STANDARD_WELD_DATA := W#16#0;
   S700_BT_CODE_2109.RBT15_STANDARD_WELD_DATA := W#16#0;
   S700_BT_CODE_2109.RBT16_STANDARD_WELD_DATA := W#16#0;
   S700_BT_CODE_2109.RBT17_STANDARD_WELD_DATA := W#16#0;
   S700_BT_CODE_2109.RBT18_STANDARD_WELD_DATA := W#16#0;
   S700_BT_CODE_2109.RBT19_STANDARD_WELD_DATA := W#16#0;
   S700_BT_CODE_2109.RBT20_STANDARD_WELD_DATA := W#16#0;
   S700_BT_CODE_2109.RBT21_STANDARD_WELD_DATA := W#16#0;
   S700_BT_CODE_2109.RBT22_STANDARD_WELD_DATA := W#16#0;
   S700_BT_CODE_2109.RBT23_STANDARD_WELD_DAT := W#16#0;
   S700_BT_CODE_2109.RBT24_STANDARD_WELD_DAT := W#16#0;
   S700_BT_CODE_2109.CHK_WORD := W#16#0;
   S700_BT_CODE_2109.TEST_TEMP[1] := B#16#0;
   S700_BT_CODE_2109.TEST_TEMP[2] := B#16#0;
   S700_BT_CODE_2109.TEST_TEMP[3] := B#16#0;
   S700_BT_CODE_2109.TEST_TEMP[4] := B#16#0;
   S700_BT_CODE_2109.TEST_TEMP[5] := B#16#0;
   S700_BT_CODE_2109.TEST_TEMP[6] := B#16#0;
   S700_BT_CODE_2109.TEST_TEMP[7] := B#16#0;
   S700_BT_CODE_2109.TEST_TEMP[8] := B#16#0;
   S700_BT_CODE_2109.TEST_TEMP[9] := B#16#0;
   S700_BT_CODE_2109.TEST_TEMP[10] := B#16#0;
   S700_BT_CODE_2109.TEST_TEMP[11] := B#16#0;
   S700_BT_CODE_2109.TEST_TEMP[12] := B#16#0;
   S700_BT_CODE_2109.TEST_TEMP[13] := B#16#0;
   S700_BT_CODE_2109.TEST_TEMP[14] := B#16#0;
   S700_BT_CODE_2109.TEST_TEMP[15] := B#16#0;
   S700_BT_CODE_2109.TEST_TEMP[16] := B#16#0;
   S700_BT_CODE_2109.TEST_TEMP[17] := B#16#0;
   S700_BT_CODE_2109.TEST_TEMP[18] := B#16#0;
   S700_BT_CODE_2109.TEST_TEMP[19] := B#16#0;
   S700_BT_CODE_2109.TEST_TEMP[20] := B#16#0;
   S700_BT_CODE_2109.TEST_TEMP[21] := B#16#0;
   S700_BT_CODE_2109.TEST_TEMP[22] := B#16#0;
   S700_BT_CODE_2109.TEST_TEMP[23] := B#16#0;
   S700_BT_CODE_2109.TEST_TEMP[24] := B#16#0;
   S700_BT_CODE_2109.TEST_TEMP[25] := B#16#0;
   S700_BT_CODE_2109.TEST_TEMP[26] := B#16#0;
   S700_BT_CODE_2109.TEST_TEMP[27] := B#16#0;
   S700_BT_CODE_2109.TEST_TEMP[28] := B#16#0;
   S700_BT_CODE_2109.TEST_TEMP[29] := B#16#0;
   S700_BT_CODE_2109.TEST_TEMP[30] := B#16#0;
   S700_BT_CODE_2109.TEST_TEMP[31] := B#16#0;
   S700_BT_CODE_2109.TEST_TEMP[32] := B#16#0;
   S700_BT_CODE_2109.TEST_TEMP[33] := B#16#0;
   S700_BT_CODE_2109.TEST_TEMP[34] := B#16#0;
   S700_BT_CODE_2109.TEST_TEMP[35] := B#16#0;
   S700_BT_CODE_2109.TEST_TEMP[36] := B#16#0;
   S700_BT_CODE_2109.TEST_TEMP[37] := B#16#0;
   S700_BT_CODE_2109.TEST_TEMP[38] := B#16#0;
   S700_BT_CODE_2109.TEST_TEMP[39] := B#16#0;
   S700_BT_CODE_2109.TEST_TEMP[40] := B#16#0;
   S700_BT_CODE_2110.STATION_MAIN := W#16#0;
   S700_BT_CODE_2110.DISTINCTION_LH_RH := W#16#0;
   S700_BT_CODE_2110.STAION_NUMBER := W#16#0;
   S700_BT_CODE_2110.BODY_TYPE_1ST := W#16#0;
   S700_BT_CODE_2110.BODY_TYPE_OPTION := W#16#0;
   S700_BT_CODE_2110.RBT1_STANDARD_WELD_DATA := W#16#0;
   S700_BT_CODE_2110.RBT2_STANDARD_WELD_DATA := W#16#0;
   S700_BT_CODE_2110.RBT3_STANDARD_WELD_DATA := W#16#0;
   S700_BT_CODE_2110.RBT4_STANDARD_WELD_DATA := W#16#0;
   S700_BT_CODE_2110.RBT5_STANDARD_WELD_DATA := W#16#0;
   S700_BT_CODE_2110.RBT6_STANDARD_WELD_DATA := W#16#0;
   S700_BT_CODE_2110.RBT7_STANDARD_WELD_DATA := W#16#0;
   S700_BT_CODE_2110.RBT8_STANDARD_WELD_DATA := W#16#0;
   S700_BT_CODE_2110.RBT9_STANDARD_WELD_DATA := W#16#0;
   S700_BT_CODE_2110.RBT10_STANDARD_WELD_DATA := W#16#0;
   S700_BT_CODE_2110.RBT11_STANDARD_WELD_DATA := W#16#0;
   S700_BT_CODE_2110.RBT12_STANDARD_WELD_DATA := W#16#0;
   S700_BT_CODE_2110.RBT13_STANDARD_WELD_DATA := W#16#0;
   S700_BT_CODE_2110.RBT14_STANDARD_WELD_DATA := W#16#0;
   S700_BT_CODE_2110.RBT15_STANDARD_WELD_DATA := W#16#0;
   S700_BT_CODE_2110.RBT16_STANDARD_WELD_DATA := W#16#0;
   S700_BT_CODE_2110.RBT17_STANDARD_WELD_DATA := W#16#0;
   S700_BT_CODE_2110.RBT18_STANDARD_WELD_DATA := W#16#0;
   S700_BT_CODE_2110.RBT19_STANDARD_WELD_DATA := W#16#0;
   S700_BT_CODE_2110.RBT20_STANDARD_WELD_DATA := W#16#0;
   S700_BT_CODE_2110.RBT21_STANDARD_WELD_DATA := W#16#0;
   S700_BT_CODE_2110.RBT22_STANDARD_WELD_DATA := W#16#0;
   S700_BT_CODE_2110.RBT23_STANDARD_WELD_DAT := W#16#0;
   S700_BT_CODE_2110.RBT24_STANDARD_WELD_DAT := W#16#0;
   S700_BT_CODE_2110.CHK_WORD := W#16#0;
   S700_BT_CODE_2110.TEST_TEMP[1] := B#16#0;
   S700_BT_CODE_2110.TEST_TEMP[2] := B#16#0;
   S700_BT_CODE_2110.TEST_TEMP[3] := B#16#0;
   S700_BT_CODE_2110.TEST_TEMP[4] := B#16#0;
   S700_BT_CODE_2110.TEST_TEMP[5] := B#16#0;
   S700_BT_CODE_2110.TEST_TEMP[6] := B#16#0;
   S700_BT_CODE_2110.TEST_TEMP[7] := B#16#0;
   S700_BT_CODE_2110.TEST_TEMP[8] := B#16#0;
   S700_BT_CODE_2110.TEST_TEMP[9] := B#16#0;
   S700_BT_CODE_2110.TEST_TEMP[10] := B#16#0;
   S700_BT_CODE_2110.TEST_TEMP[11] := B#16#0;
   S700_BT_CODE_2110.TEST_TEMP[12] := B#16#0;
   S700_BT_CODE_2110.TEST_TEMP[13] := B#16#0;
   S700_BT_CODE_2110.TEST_TEMP[14] := B#16#0;
   S700_BT_CODE_2110.TEST_TEMP[15] := B#16#0;
   S700_BT_CODE_2110.TEST_TEMP[16] := B#16#0;
   S700_BT_CODE_2110.TEST_TEMP[17] := B#16#0;
   S700_BT_CODE_2110.TEST_TEMP[18] := B#16#0;
   S700_BT_CODE_2110.TEST_TEMP[19] := B#16#0;
   S700_BT_CODE_2110.TEST_TEMP[20] := B#16#0;
   S700_BT_CODE_2110.TEST_TEMP[21] := B#16#0;
   S700_BT_CODE_2110.TEST_TEMP[22] := B#16#0;
   S700_BT_CODE_2110.TEST_TEMP[23] := B#16#0;
   S700_BT_CODE_2110.TEST_TEMP[24] := B#16#0;
   S700_BT_CODE_2110.TEST_TEMP[25] := B#16#0;
   S700_BT_CODE_2110.TEST_TEMP[26] := B#16#0;
   S700_BT_CODE_2110.TEST_TEMP[27] := B#16#0;
   S700_BT_CODE_2110.TEST_TEMP[28] := B#16#0;
   S700_BT_CODE_2110.TEST_TEMP[29] := B#16#0;
   S700_BT_CODE_2110.TEST_TEMP[30] := B#16#0;
   S700_BT_CODE_2110.TEST_TEMP[31] := B#16#0;
   S700_BT_CODE_2110.TEST_TEMP[32] := B#16#0;
   S700_BT_CODE_2110.TEST_TEMP[33] := B#16#0;
   S700_BT_CODE_2110.TEST_TEMP[34] := B#16#0;
   S700_BT_CODE_2110.TEST_TEMP[35] := B#16#0;
   S700_BT_CODE_2110.TEST_TEMP[36] := B#16#0;
   S700_BT_CODE_2110.TEST_TEMP[37] := B#16#0;
   S700_BT_CODE_2110.TEST_TEMP[38] := B#16#0;
   S700_BT_CODE_2110.TEST_TEMP[39] := B#16#0;
   S700_BT_CODE_2110.TEST_TEMP[40] := B#16#0;
   S700_BT_CODE_2111.STATION_MAIN := W#16#0;
   S700_BT_CODE_2111.DISTINCTION_LH_RH := W#16#0;
   S700_BT_CODE_2111.STAION_NUMBER := W#16#0;
   S700_BT_CODE_2111.BODY_TYPE_1ST := W#16#0;
   S700_BT_CODE_2111.BODY_TYPE_OPTION := W#16#0;
   S700_BT_CODE_2111.RBT1_STANDARD_WELD_DATA := W#16#0;
   S700_BT_CODE_2111.RBT2_STANDARD_WELD_DATA := W#16#0;
   S700_BT_CODE_2111.RBT3_STANDARD_WELD_DATA := W#16#0;
   S700_BT_CODE_2111.RBT4_STANDARD_WELD_DATA := W#16#0;
   S700_BT_CODE_2111.RBT5_STANDARD_WELD_DATA := W#16#0;
   S700_BT_CODE_2111.RBT6_STANDARD_WELD_DATA := W#16#0;
   S700_BT_CODE_2111.RBT7_STANDARD_WELD_DATA := W#16#0;
   S700_BT_CODE_2111.RBT8_STANDARD_WELD_DATA := W#16#0;
   S700_BT_CODE_2111.RBT9_STANDARD_WELD_DATA := W#16#0;
   S700_BT_CODE_2111.RBT10_STANDARD_WELD_DATA := W#16#0;
   S700_BT_CODE_2111.RBT11_STANDARD_WELD_DATA := W#16#0;
   S700_BT_CODE_2111.RBT12_STANDARD_WELD_DATA := W#16#0;
   S700_BT_CODE_2111.RBT13_STANDARD_WELD_DATA := W#16#0;
   S700_BT_CODE_2111.RBT14_STANDARD_WELD_DATA := W#16#0;
   S700_BT_CODE_2111.RBT15_STANDARD_WELD_DATA := W#16#0;
   S700_BT_CODE_2111.RBT16_STANDARD_WELD_DATA := W#16#0;
   S700_BT_CODE_2111.RBT17_STANDARD_WELD_DATA := W#16#0;
   S700_BT_CODE_2111.RBT18_STANDARD_WELD_DATA := W#16#0;
   S700_BT_CODE_2111.RBT19_STANDARD_WELD_DATA := W#16#0;
   S700_BT_CODE_2111.RBT20_STANDARD_WELD_DATA := W#16#0;
   S700_BT_CODE_2111.RBT21_STANDARD_WELD_DATA := W#16#0;
   S700_BT_CODE_2111.RBT22_STANDARD_WELD_DATA := W#16#0;
   S700_BT_CODE_2111.RBT23_STANDARD_WELD_DAT := W#16#0;
   S700_BT_CODE_2111.RBT24_STANDARD_WELD_DAT := W#16#0;
   S700_BT_CODE_2111.CHK_WORD := W#16#0;
   S700_BT_CODE_2111.TEST_TEMP[1] := B#16#0;
   S700_BT_CODE_2111.TEST_TEMP[2] := B#16#0;
   S700_BT_CODE_2111.TEST_TEMP[3] := B#16#0;
   S700_BT_CODE_2111.TEST_TEMP[4] := B#16#0;
   S700_BT_CODE_2111.TEST_TEMP[5] := B#16#0;
   S700_BT_CODE_2111.TEST_TEMP[6] := B#16#0;
   S700_BT_CODE_2111.TEST_TEMP[7] := B#16#0;
   S700_BT_CODE_2111.TEST_TEMP[8] := B#16#0;
   S700_BT_CODE_2111.TEST_TEMP[9] := B#16#0;
   S700_BT_CODE_2111.TEST_TEMP[10] := B#16#0;
   S700_BT_CODE_2111.TEST_TEMP[11] := B#16#0;
   S700_BT_CODE_2111.TEST_TEMP[12] := B#16#0;
   S700_BT_CODE_2111.TEST_TEMP[13] := B#16#0;
   S700_BT_CODE_2111.TEST_TEMP[14] := B#16#0;
   S700_BT_CODE_2111.TEST_TEMP[15] := B#16#0;
   S700_BT_CODE_2111.TEST_TEMP[16] := B#16#0;
   S700_BT_CODE_2111.TEST_TEMP[17] := B#16#0;
   S700_BT_CODE_2111.TEST_TEMP[18] := B#16#0;
   S700_BT_CODE_2111.TEST_TEMP[19] := B#16#0;
   S700_BT_CODE_2111.TEST_TEMP[20] := B#16#0;
   S700_BT_CODE_2111.TEST_TEMP[21] := B#16#0;
   S700_BT_CODE_2111.TEST_TEMP[22] := B#16#0;
   S700_BT_CODE_2111.TEST_TEMP[23] := B#16#0;
   S700_BT_CODE_2111.TEST_TEMP[24] := B#16#0;
   S700_BT_CODE_2111.TEST_TEMP[25] := B#16#0;
   S700_BT_CODE_2111.TEST_TEMP[26] := B#16#0;
   S700_BT_CODE_2111.TEST_TEMP[27] := B#16#0;
   S700_BT_CODE_2111.TEST_TEMP[28] := B#16#0;
   S700_BT_CODE_2111.TEST_TEMP[29] := B#16#0;
   S700_BT_CODE_2111.TEST_TEMP[30] := B#16#0;
   S700_BT_CODE_2111.TEST_TEMP[31] := B#16#0;
   S700_BT_CODE_2111.TEST_TEMP[32] := B#16#0;
   S700_BT_CODE_2111.TEST_TEMP[33] := B#16#0;
   S700_BT_CODE_2111.TEST_TEMP[34] := B#16#0;
   S700_BT_CODE_2111.TEST_TEMP[35] := B#16#0;
   S700_BT_CODE_2111.TEST_TEMP[36] := B#16#0;
   S700_BT_CODE_2111.TEST_TEMP[37] := B#16#0;
   S700_BT_CODE_2111.TEST_TEMP[38] := B#16#0;
   S700_BT_CODE_2111.TEST_TEMP[39] := B#16#0;
   S700_BT_CODE_2111.TEST_TEMP[40] := B#16#0;
   S700_BT_CODE_2112.STATION_MAIN := W#16#0;
   S700_BT_CODE_2112.DISTINCTION_LH_RH := W#16#0;
   S700_BT_CODE_2112.STAION_NUMBER := W#16#0;
   S700_BT_CODE_2112.BODY_TYPE_1ST := W#16#0;
   S700_BT_CODE_2112.BODY_TYPE_OPTION := W#16#0;
   S700_BT_CODE_2112.RBT1_STANDARD_WELD_DATA := W#16#0;
   S700_BT_CODE_2112.RBT2_STANDARD_WELD_DATA := W#16#0;
   S700_BT_CODE_2112.RBT3_STANDARD_WELD_DATA := W#16#0;
   S700_BT_CODE_2112.RBT4_STANDARD_WELD_DATA := W#16#0;
   S700_BT_CODE_2112.RBT5_STANDARD_WELD_DATA := W#16#0;
   S700_BT_CODE_2112.RBT6_STANDARD_WELD_DATA := W#16#0;
   S700_BT_CODE_2112.RBT7_STANDARD_WELD_DATA := W#16#0;
   S700_BT_CODE_2112.RBT8_STANDARD_WELD_DATA := W#16#0;
   S700_BT_CODE_2112.RBT9_STANDARD_WELD_DATA := W#16#0;
   S700_BT_CODE_2112.RBT10_STANDARD_WELD_DATA := W#16#0;
   S700_BT_CODE_2112.RBT11_STANDARD_WELD_DATA := W#16#0;
   S700_BT_CODE_2112.RBT12_STANDARD_WELD_DATA := W#16#0;
   S700_BT_CODE_2112.RBT13_STANDARD_WELD_DATA := W#16#0;
   S700_BT_CODE_2112.RBT14_STANDARD_WELD_DATA := W#16#0;
   S700_BT_CODE_2112.RBT15_STANDARD_WELD_DATA := W#16#0;
   S700_BT_CODE_2112.RBT16_STANDARD_WELD_DATA := W#16#0;
   S700_BT_CODE_2112.RBT17_STANDARD_WELD_DATA := W#16#0;
   S700_BT_CODE_2112.RBT18_STANDARD_WELD_DATA := W#16#0;
   S700_BT_CODE_2112.RBT19_STANDARD_WELD_DATA := W#16#0;
   S700_BT_CODE_2112.RBT20_STANDARD_WELD_DATA := W#16#0;
   S700_BT_CODE_2112.RBT21_STANDARD_WELD_DATA := W#16#0;
   S700_BT_CODE_2112.RBT22_STANDARD_WELD_DATA := W#16#0;
   S700_BT_CODE_2112.RBT23_STANDARD_WELD_DAT := W#16#0;
   S700_BT_CODE_2112.RBT24_STANDARD_WELD_DAT := W#16#0;
   S700_BT_CODE_2112.CHK_WORD := W#16#0;
   S700_BT_CODE_2112.TEST_TEMP[1] := B#16#0;
   S700_BT_CODE_2112.TEST_TEMP[2] := B#16#0;
   S700_BT_CODE_2112.TEST_TEMP[3] := B#16#0;
   S700_BT_CODE_2112.TEST_TEMP[4] := B#16#0;
   S700_BT_CODE_2112.TEST_TEMP[5] := B#16#0;
   S700_BT_CODE_2112.TEST_TEMP[6] := B#16#0;
   S700_BT_CODE_2112.TEST_TEMP[7] := B#16#0;
   S700_BT_CODE_2112.TEST_TEMP[8] := B#16#0;
   S700_BT_CODE_2112.TEST_TEMP[9] := B#16#0;
   S700_BT_CODE_2112.TEST_TEMP[10] := B#16#0;
   S700_BT_CODE_2112.TEST_TEMP[11] := B#16#0;
   S700_BT_CODE_2112.TEST_TEMP[12] := B#16#0;
   S700_BT_CODE_2112.TEST_TEMP[13] := B#16#0;
   S700_BT_CODE_2112.TEST_TEMP[14] := B#16#0;
   S700_BT_CODE_2112.TEST_TEMP[15] := B#16#0;
   S700_BT_CODE_2112.TEST_TEMP[16] := B#16#0;
   S700_BT_CODE_2112.TEST_TEMP[17] := B#16#0;
   S700_BT_CODE_2112.TEST_TEMP[18] := B#16#0;
   S700_BT_CODE_2112.TEST_TEMP[19] := B#16#0;
   S700_BT_CODE_2112.TEST_TEMP[20] := B#16#0;
   S700_BT_CODE_2112.TEST_TEMP[21] := B#16#0;
   S700_BT_CODE_2112.TEST_TEMP[22] := B#16#0;
   S700_BT_CODE_2112.TEST_TEMP[23] := B#16#0;
   S700_BT_CODE_2112.TEST_TEMP[24] := B#16#0;
   S700_BT_CODE_2112.TEST_TEMP[25] := B#16#0;
   S700_BT_CODE_2112.TEST_TEMP[26] := B#16#0;
   S700_BT_CODE_2112.TEST_TEMP[27] := B#16#0;
   S700_BT_CODE_2112.TEST_TEMP[28] := B#16#0;
   S700_BT_CODE_2112.TEST_TEMP[29] := B#16#0;
   S700_BT_CODE_2112.TEST_TEMP[30] := B#16#0;
   S700_BT_CODE_2112.TEST_TEMP[31] := B#16#0;
   S700_BT_CODE_2112.TEST_TEMP[32] := B#16#0;
   S700_BT_CODE_2112.TEST_TEMP[33] := B#16#0;
   S700_BT_CODE_2112.TEST_TEMP[34] := B#16#0;
   S700_BT_CODE_2112.TEST_TEMP[35] := B#16#0;
   S700_BT_CODE_2112.TEST_TEMP[36] := B#16#0;
   S700_BT_CODE_2112.TEST_TEMP[37] := B#16#0;
   S700_BT_CODE_2112.TEST_TEMP[38] := B#16#0;
   S700_BT_CODE_2112.TEST_TEMP[39] := B#16#0;
   S700_BT_CODE_2112.TEST_TEMP[40] := B#16#0;
   S700_BT_CODE_2113.STATION_MAIN := W#16#0;
   S700_BT_CODE_2113.DISTINCTION_LH_RH := W#16#0;
   S700_BT_CODE_2113.STAION_NUMBER := W#16#0;
   S700_BT_CODE_2113.BODY_TYPE_1ST := W#16#0;
   S700_BT_CODE_2113.BODY_TYPE_OPTION := W#16#0;
   S700_BT_CODE_2113.RBT1_STANDARD_WELD_DATA := W#16#0;
   S700_BT_CODE_2113.RBT2_STANDARD_WELD_DATA := W#16#0;
   S700_BT_CODE_2113.RBT3_STANDARD_WELD_DATA := W#16#0;
   S700_BT_CODE_2113.RBT4_STANDARD_WELD_DATA := W#16#0;
   S700_BT_CODE_2113.RBT5_STANDARD_WELD_DATA := W#16#0;
   S700_BT_CODE_2113.RBT6_STANDARD_WELD_DATA := W#16#0;
   S700_BT_CODE_2113.RBT7_STANDARD_WELD_DATA := W#16#0;
   S700_BT_CODE_2113.RBT8_STANDARD_WELD_DATA := W#16#0;
   S700_BT_CODE_2113.RBT9_STANDARD_WELD_DATA := W#16#0;
   S700_BT_CODE_2113.RBT10_STANDARD_WELD_DATA := W#16#0;
   S700_BT_CODE_2113.RBT11_STANDARD_WELD_DATA := W#16#0;
   S700_BT_CODE_2113.RBT12_STANDARD_WELD_DATA := W#16#0;
   S700_BT_CODE_2113.RBT13_STANDARD_WELD_DATA := W#16#0;
   S700_BT_CODE_2113.RBT14_STANDARD_WELD_DATA := W#16#0;
   S700_BT_CODE_2113.RBT15_STANDARD_WELD_DATA := W#16#0;
   S700_BT_CODE_2113.RBT16_STANDARD_WELD_DATA := W#16#0;
   S700_BT_CODE_2113.RBT17_STANDARD_WELD_DATA := W#16#0;
   S700_BT_CODE_2113.RBT18_STANDARD_WELD_DATA := W#16#0;
   S700_BT_CODE_2113.RBT19_STANDARD_WELD_DATA := W#16#0;
   S700_BT_CODE_2113.RBT20_STANDARD_WELD_DATA := W#16#0;
   S700_BT_CODE_2113.RBT21_STANDARD_WELD_DATA := W#16#0;
   S700_BT_CODE_2113.RBT22_STANDARD_WELD_DATA := W#16#0;
   S700_BT_CODE_2113.RBT23_STANDARD_WELD_DAT := W#16#0;
   S700_BT_CODE_2113.RBT24_STANDARD_WELD_DAT := W#16#0;
   S700_BT_CODE_2113.CHK_WORD := W#16#0;
   S700_BT_CODE_2113.TEST_TEMP[1] := B#16#0;
   S700_BT_CODE_2113.TEST_TEMP[2] := B#16#0;
   S700_BT_CODE_2113.TEST_TEMP[3] := B#16#0;
   S700_BT_CODE_2113.TEST_TEMP[4] := B#16#0;
   S700_BT_CODE_2113.TEST_TEMP[5] := B#16#0;
   S700_BT_CODE_2113.TEST_TEMP[6] := B#16#0;
   S700_BT_CODE_2113.TEST_TEMP[7] := B#16#0;
   S700_BT_CODE_2113.TEST_TEMP[8] := B#16#0;
   S700_BT_CODE_2113.TEST_TEMP[9] := B#16#0;
   S700_BT_CODE_2113.TEST_TEMP[10] := B#16#0;
   S700_BT_CODE_2113.TEST_TEMP[11] := B#16#0;
   S700_BT_CODE_2113.TEST_TEMP[12] := B#16#0;
   S700_BT_CODE_2113.TEST_TEMP[13] := B#16#0;
   S700_BT_CODE_2113.TEST_TEMP[14] := B#16#0;
   S700_BT_CODE_2113.TEST_TEMP[15] := B#16#0;
   S700_BT_CODE_2113.TEST_TEMP[16] := B#16#0;
   S700_BT_CODE_2113.TEST_TEMP[17] := B#16#0;
   S700_BT_CODE_2113.TEST_TEMP[18] := B#16#0;
   S700_BT_CODE_2113.TEST_TEMP[19] := B#16#0;
   S700_BT_CODE_2113.TEST_TEMP[20] := B#16#0;
   S700_BT_CODE_2113.TEST_TEMP[21] := B#16#0;
   S700_BT_CODE_2113.TEST_TEMP[22] := B#16#0;
   S700_BT_CODE_2113.TEST_TEMP[23] := B#16#0;
   S700_BT_CODE_2113.TEST_TEMP[24] := B#16#0;
   S700_BT_CODE_2113.TEST_TEMP[25] := B#16#0;
   S700_BT_CODE_2113.TEST_TEMP[26] := B#16#0;
   S700_BT_CODE_2113.TEST_TEMP[27] := B#16#0;
   S700_BT_CODE_2113.TEST_TEMP[28] := B#16#0;
   S700_BT_CODE_2113.TEST_TEMP[29] := B#16#0;
   S700_BT_CODE_2113.TEST_TEMP[30] := B#16#0;
   S700_BT_CODE_2113.TEST_TEMP[31] := B#16#0;
   S700_BT_CODE_2113.TEST_TEMP[32] := B#16#0;
   S700_BT_CODE_2113.TEST_TEMP[33] := B#16#0;
   S700_BT_CODE_2113.TEST_TEMP[34] := B#16#0;
   S700_BT_CODE_2113.TEST_TEMP[35] := B#16#0;
   S700_BT_CODE_2113.TEST_TEMP[36] := B#16#0;
   S700_BT_CODE_2113.TEST_TEMP[37] := B#16#0;
   S700_BT_CODE_2113.TEST_TEMP[38] := B#16#0;
   S700_BT_CODE_2113.TEST_TEMP[39] := B#16#0;
   S700_BT_CODE_2113.TEST_TEMP[40] := B#16#0;
   S700_BT_CODE_2114.STATION_MAIN := W#16#0;
   S700_BT_CODE_2114.DISTINCTION_LH_RH := W#16#0;
   S700_BT_CODE_2114.STAION_NUMBER := W#16#0;
   S700_BT_CODE_2114.BODY_TYPE_1ST := W#16#0;
   S700_BT_CODE_2114.BODY_TYPE_OPTION := W#16#0;
   S700_BT_CODE_2114.RBT1_STANDARD_WELD_DATA := W#16#0;
   S700_BT_CODE_2114.RBT2_STANDARD_WELD_DATA := W#16#0;
   S700_BT_CODE_2114.RBT3_STANDARD_WELD_DATA := W#16#0;
   S700_BT_CODE_2114.RBT4_STANDARD_WELD_DATA := W#16#0;
   S700_BT_CODE_2114.RBT5_STANDARD_WELD_DATA := W#16#0;
   S700_BT_CODE_2114.RBT6_STANDARD_WELD_DATA := W#16#0;
   S700_BT_CODE_2114.RBT7_STANDARD_WELD_DATA := W#16#0;
   S700_BT_CODE_2114.RBT8_STANDARD_WELD_DATA := W#16#0;
   S700_BT_CODE_2114.RBT9_STANDARD_WELD_DATA := W#16#0;
   S700_BT_CODE_2114.RBT10_STANDARD_WELD_DATA := W#16#0;
   S700_BT_CODE_2114.RBT11_STANDARD_WELD_DATA := W#16#0;
   S700_BT_CODE_2114.RBT12_STANDARD_WELD_DATA := W#16#0;
   S700_BT_CODE_2114.RBT13_STANDARD_WELD_DATA := W#16#0;
   S700_BT_CODE_2114.RBT14_STANDARD_WELD_DATA := W#16#0;
   S700_BT_CODE_2114.RBT15_STANDARD_WELD_DATA := W#16#0;
   S700_BT_CODE_2114.RBT16_STANDARD_WELD_DATA := W#16#0;
   S700_BT_CODE_2114.RBT17_STANDARD_WELD_DATA := W#16#0;
   S700_BT_CODE_2114.RBT18_STANDARD_WELD_DATA := W#16#0;
   S700_BT_CODE_2114.RBT19_STANDARD_WELD_DATA := W#16#0;
   S700_BT_CODE_2114.RBT20_STANDARD_WELD_DATA := W#16#0;
   S700_BT_CODE_2114.RBT21_STANDARD_WELD_DATA := W#16#0;
   S700_BT_CODE_2114.RBT22_STANDARD_WELD_DATA := W#16#0;
   S700_BT_CODE_2114.RBT23_STANDARD_WELD_DAT := W#16#0;
   S700_BT_CODE_2114.RBT24_STANDARD_WELD_DAT := W#16#0;
   S700_BT_CODE_2114.CHK_WORD := W#16#0;
   S700_BT_CODE_2114.TEST_TEMP[1] := B#16#0;
   S700_BT_CODE_2114.TEST_TEMP[2] := B#16#0;
   S700_BT_CODE_2114.TEST_TEMP[3] := B#16#0;
   S700_BT_CODE_2114.TEST_TEMP[4] := B#16#0;
   S700_BT_CODE_2114.TEST_TEMP[5] := B#16#0;
   S700_BT_CODE_2114.TEST_TEMP[6] := B#16#0;
   S700_BT_CODE_2114.TEST_TEMP[7] := B#16#0;
   S700_BT_CODE_2114.TEST_TEMP[8] := B#16#0;
   S700_BT_CODE_2114.TEST_TEMP[9] := B#16#0;
   S700_BT_CODE_2114.TEST_TEMP[10] := B#16#0;
   S700_BT_CODE_2114.TEST_TEMP[11] := B#16#0;
   S700_BT_CODE_2114.TEST_TEMP[12] := B#16#0;
   S700_BT_CODE_2114.TEST_TEMP[13] := B#16#0;
   S700_BT_CODE_2114.TEST_TEMP[14] := B#16#0;
   S700_BT_CODE_2114.TEST_TEMP[15] := B#16#0;
   S700_BT_CODE_2114.TEST_TEMP[16] := B#16#0;
   S700_BT_CODE_2114.TEST_TEMP[17] := B#16#0;
   S700_BT_CODE_2114.TEST_TEMP[18] := B#16#0;
   S700_BT_CODE_2114.TEST_TEMP[19] := B#16#0;
   S700_BT_CODE_2114.TEST_TEMP[20] := B#16#0;
   S700_BT_CODE_2114.TEST_TEMP[21] := B#16#0;
   S700_BT_CODE_2114.TEST_TEMP[22] := B#16#0;
   S700_BT_CODE_2114.TEST_TEMP[23] := B#16#0;
   S700_BT_CODE_2114.TEST_TEMP[24] := B#16#0;
   S700_BT_CODE_2114.TEST_TEMP[25] := B#16#0;
   S700_BT_CODE_2114.TEST_TEMP[26] := B#16#0;
   S700_BT_CODE_2114.TEST_TEMP[27] := B#16#0;
   S700_BT_CODE_2114.TEST_TEMP[28] := B#16#0;
   S700_BT_CODE_2114.TEST_TEMP[29] := B#16#0;
   S700_BT_CODE_2114.TEST_TEMP[30] := B#16#0;
   S700_BT_CODE_2114.TEST_TEMP[31] := B#16#0;
   S700_BT_CODE_2114.TEST_TEMP[32] := B#16#0;
   S700_BT_CODE_2114.TEST_TEMP[33] := B#16#0;
   S700_BT_CODE_2114.TEST_TEMP[34] := B#16#0;
   S700_BT_CODE_2114.TEST_TEMP[35] := B#16#0;
   S700_BT_CODE_2114.TEST_TEMP[36] := B#16#0;
   S700_BT_CODE_2114.TEST_TEMP[37] := B#16#0;
   S700_BT_CODE_2114.TEST_TEMP[38] := B#16#0;
   S700_BT_CODE_2114.TEST_TEMP[39] := B#16#0;
   S700_BT_CODE_2114.TEST_TEMP[40] := B#16#0;
   S700_BT_CODE_2115.STATION_MAIN := W#16#0;
   S700_BT_CODE_2115.DISTINCTION_LH_RH := W#16#0;
   S700_BT_CODE_2115.STAION_NUMBER := W#16#0;
   S700_BT_CODE_2115.BODY_TYPE_1ST := W#16#0;
   S700_BT_CODE_2115.BODY_TYPE_OPTION := W#16#0;
   S700_BT_CODE_2115.RBT1_STANDARD_WELD_DATA := W#16#0;
   S700_BT_CODE_2115.RBT2_STANDARD_WELD_DATA := W#16#0;
   S700_BT_CODE_2115.RBT3_STANDARD_WELD_DATA := W#16#0;
   S700_BT_CODE_2115.RBT4_STANDARD_WELD_DATA := W#16#0;
   S700_BT_CODE_2115.RBT5_STANDARD_WELD_DATA := W#16#0;
   S700_BT_CODE_2115.RBT6_STANDARD_WELD_DATA := W#16#0;
   S700_BT_CODE_2115.RBT7_STANDARD_WELD_DATA := W#16#0;
   S700_BT_CODE_2115.RBT8_STANDARD_WELD_DATA := W#16#0;
   S700_BT_CODE_2115.RBT9_STANDARD_WELD_DATA := W#16#0;
   S700_BT_CODE_2115.RBT10_STANDARD_WELD_DATA := W#16#0;
   S700_BT_CODE_2115.RBT11_STANDARD_WELD_DATA := W#16#0;
   S700_BT_CODE_2115.RBT12_STANDARD_WELD_DATA := W#16#0;
   S700_BT_CODE_2115.RBT13_STANDARD_WELD_DATA := W#16#0;
   S700_BT_CODE_2115.RBT14_STANDARD_WELD_DATA := W#16#0;
   S700_BT_CODE_2115.RBT15_STANDARD_WELD_DATA := W#16#0;
   S700_BT_CODE_2115.RBT16_STANDARD_WELD_DATA := W#16#0;
   S700_BT_CODE_2115.RBT17_STANDARD_WELD_DATA := W#16#0;
   S700_BT_CODE_2115.RBT18_STANDARD_WELD_DATA := W#16#0;
   S700_BT_CODE_2115.RBT19_STANDARD_WELD_DATA := W#16#0;
   S700_BT_CODE_2115.RBT20_STANDARD_WELD_DATA := W#16#0;
   S700_BT_CODE_2115.RBT21_STANDARD_WELD_DATA := W#16#0;
   S700_BT_CODE_2115.RBT22_STANDARD_WELD_DATA := W#16#0;
   S700_BT_CODE_2115.RBT23_STANDARD_WELD_DAT := W#16#0;
   S700_BT_CODE_2115.RBT24_STANDARD_WELD_DAT := W#16#0;
   S700_BT_CODE_2115.CHK_WORD := W#16#0;
   S700_BT_CODE_2115.TEST_TEMP[1] := B#16#0;
   S700_BT_CODE_2115.TEST_TEMP[2] := B#16#0;
   S700_BT_CODE_2115.TEST_TEMP[3] := B#16#0;
   S700_BT_CODE_2115.TEST_TEMP[4] := B#16#0;
   S700_BT_CODE_2115.TEST_TEMP[5] := B#16#0;
   S700_BT_CODE_2115.TEST_TEMP[6] := B#16#0;
   S700_BT_CODE_2115.TEST_TEMP[7] := B#16#0;
   S700_BT_CODE_2115.TEST_TEMP[8] := B#16#0;
   S700_BT_CODE_2115.TEST_TEMP[9] := B#16#0;
   S700_BT_CODE_2115.TEST_TEMP[10] := B#16#0;
   S700_BT_CODE_2115.TEST_TEMP[11] := B#16#0;
   S700_BT_CODE_2115.TEST_TEMP[12] := B#16#0;
   S700_BT_CODE_2115.TEST_TEMP[13] := B#16#0;
   S700_BT_CODE_2115.TEST_TEMP[14] := B#16#0;
   S700_BT_CODE_2115.TEST_TEMP[15] := B#16#0;
   S700_BT_CODE_2115.TEST_TEMP[16] := B#16#0;
   S700_BT_CODE_2115.TEST_TEMP[17] := B#16#0;
   S700_BT_CODE_2115.TEST_TEMP[18] := B#16#0;
   S700_BT_CODE_2115.TEST_TEMP[19] := B#16#0;
   S700_BT_CODE_2115.TEST_TEMP[20] := B#16#0;
   S700_BT_CODE_2115.TEST_TEMP[21] := B#16#0;
   S700_BT_CODE_2115.TEST_TEMP[22] := B#16#0;
   S700_BT_CODE_2115.TEST_TEMP[23] := B#16#0;
   S700_BT_CODE_2115.TEST_TEMP[24] := B#16#0;
   S700_BT_CODE_2115.TEST_TEMP[25] := B#16#0;
   S700_BT_CODE_2115.TEST_TEMP[26] := B#16#0;
   S700_BT_CODE_2115.TEST_TEMP[27] := B#16#0;
   S700_BT_CODE_2115.TEST_TEMP[28] := B#16#0;
   S700_BT_CODE_2115.TEST_TEMP[29] := B#16#0;
   S700_BT_CODE_2115.TEST_TEMP[30] := B#16#0;
   S700_BT_CODE_2115.TEST_TEMP[31] := B#16#0;
   S700_BT_CODE_2115.TEST_TEMP[32] := B#16#0;
   S700_BT_CODE_2115.TEST_TEMP[33] := B#16#0;
   S700_BT_CODE_2115.TEST_TEMP[34] := B#16#0;
   S700_BT_CODE_2115.TEST_TEMP[35] := B#16#0;
   S700_BT_CODE_2115.TEST_TEMP[36] := B#16#0;
   S700_BT_CODE_2115.TEST_TEMP[37] := B#16#0;
   S700_BT_CODE_2115.TEST_TEMP[38] := B#16#0;
   S700_BT_CODE_2115.TEST_TEMP[39] := B#16#0;
   S700_BT_CODE_2115.TEST_TEMP[40] := B#16#0;
   S700_BT_CODE_2116.STATION_MAIN := W#16#0;
   S700_BT_CODE_2116.DISTINCTION_LH_RH := W#16#0;
   S700_BT_CODE_2116.STAION_NUMBER := W#16#0;
   S700_BT_CODE_2116.BODY_TYPE_1ST := W#16#0;
   S700_BT_CODE_2116.BODY_TYPE_OPTION := W#16#0;
   S700_BT_CODE_2116.RBT1_STANDARD_WELD_DATA := W#16#0;
   S700_BT_CODE_2116.RBT2_STANDARD_WELD_DATA := W#16#0;
   S700_BT_CODE_2116.RBT3_STANDARD_WELD_DATA := W#16#0;
   S700_BT_CODE_2116.RBT4_STANDARD_WELD_DATA := W#16#0;
   S700_BT_CODE_2116.RBT5_STANDARD_WELD_DATA := W#16#0;
   S700_BT_CODE_2116.RBT6_STANDARD_WELD_DATA := W#16#0;
   S700_BT_CODE_2116.RBT7_STANDARD_WELD_DATA := W#16#0;
   S700_BT_CODE_2116.RBT8_STANDARD_WELD_DATA := W#16#0;
   S700_BT_CODE_2116.RBT9_STANDARD_WELD_DATA := W#16#0;
   S700_BT_CODE_2116.RBT10_STANDARD_WELD_DATA := W#16#0;
   S700_BT_CODE_2116.RBT11_STANDARD_WELD_DATA := W#16#0;
   S700_BT_CODE_2116.RBT12_STANDARD_WELD_DATA := W#16#0;
   S700_BT_CODE_2116.RBT13_STANDARD_WELD_DATA := W#16#0;
   S700_BT_CODE_2116.RBT14_STANDARD_WELD_DATA := W#16#0;
   S700_BT_CODE_2116.RBT15_STANDARD_WELD_DATA := W#16#0;
   S700_BT_CODE_2116.RBT16_STANDARD_WELD_DATA := W#16#0;
   S700_BT_CODE_2116.RBT17_STANDARD_WELD_DATA := W#16#0;
   S700_BT_CODE_2116.RBT18_STANDARD_WELD_DATA := W#16#0;
   S700_BT_CODE_2116.RBT19_STANDARD_WELD_DATA := W#16#0;
   S700_BT_CODE_2116.RBT20_STANDARD_WELD_DATA := W#16#0;
   S700_BT_CODE_2116.RBT21_STANDARD_WELD_DATA := W#16#0;
   S700_BT_CODE_2116.RBT22_STANDARD_WELD_DATA := W#16#0;
   S700_BT_CODE_2116.RBT23_STANDARD_WELD_DAT := W#16#0;
   S700_BT_CODE_2116.RBT24_STANDARD_WELD_DAT := W#16#0;
   S700_BT_CODE_2116.CHK_WORD := W#16#0;
   S700_BT_CODE_2116.TEST_TEMP[1] := B#16#0;
   S700_BT_CODE_2116.TEST_TEMP[2] := B#16#0;
   S700_BT_CODE_2116.TEST_TEMP[3] := B#16#0;
   S700_BT_CODE_2116.TEST_TEMP[4] := B#16#0;
   S700_BT_CODE_2116.TEST_TEMP[5] := B#16#0;
   S700_BT_CODE_2116.TEST_TEMP[6] := B#16#0;
   S700_BT_CODE_2116.TEST_TEMP[7] := B#16#0;
   S700_BT_CODE_2116.TEST_TEMP[8] := B#16#0;
   S700_BT_CODE_2116.TEST_TEMP[9] := B#16#0;
   S700_BT_CODE_2116.TEST_TEMP[10] := B#16#0;
   S700_BT_CODE_2116.TEST_TEMP[11] := B#16#0;
   S700_BT_CODE_2116.TEST_TEMP[12] := B#16#0;
   S700_BT_CODE_2116.TEST_TEMP[13] := B#16#0;
   S700_BT_CODE_2116.TEST_TEMP[14] := B#16#0;
   S700_BT_CODE_2116.TEST_TEMP[15] := B#16#0;
   S700_BT_CODE_2116.TEST_TEMP[16] := B#16#0;
   S700_BT_CODE_2116.TEST_TEMP[17] := B#16#0;
   S700_BT_CODE_2116.TEST_TEMP[18] := B#16#0;
   S700_BT_CODE_2116.TEST_TEMP[19] := B#16#0;
   S700_BT_CODE_2116.TEST_TEMP[20] := B#16#0;
   S700_BT_CODE_2116.TEST_TEMP[21] := B#16#0;
   S700_BT_CODE_2116.TEST_TEMP[22] := B#16#0;
   S700_BT_CODE_2116.TEST_TEMP[23] := B#16#0;
   S700_BT_CODE_2116.TEST_TEMP[24] := B#16#0;
   S700_BT_CODE_2116.TEST_TEMP[25] := B#16#0;
   S700_BT_CODE_2116.TEST_TEMP[26] := B#16#0;
   S700_BT_CODE_2116.TEST_TEMP[27] := B#16#0;
   S700_BT_CODE_2116.TEST_TEMP[28] := B#16#0;
   S700_BT_CODE_2116.TEST_TEMP[29] := B#16#0;
   S700_BT_CODE_2116.TEST_TEMP[30] := B#16#0;
   S700_BT_CODE_2116.TEST_TEMP[31] := B#16#0;
   S700_BT_CODE_2116.TEST_TEMP[32] := B#16#0;
   S700_BT_CODE_2116.TEST_TEMP[33] := B#16#0;
   S700_BT_CODE_2116.TEST_TEMP[34] := B#16#0;
   S700_BT_CODE_2116.TEST_TEMP[35] := B#16#0;
   S700_BT_CODE_2116.TEST_TEMP[36] := B#16#0;
   S700_BT_CODE_2116.TEST_TEMP[37] := B#16#0;
   S700_BT_CODE_2116.TEST_TEMP[38] := B#16#0;
   S700_BT_CODE_2116.TEST_TEMP[39] := B#16#0;
   S700_BT_CODE_2116.TEST_TEMP[40] := B#16#0;
   S700_BT_CODE_2117.STATION_MAIN := W#16#0;
   S700_BT_CODE_2117.DISTINCTION_LH_RH := W#16#0;
   S700_BT_CODE_2117.STAION_NUMBER := W#16#0;
   S700_BT_CODE_2117.BODY_TYPE_1ST := W#16#0;
   S700_BT_CODE_2117.BODY_TYPE_OPTION := W#16#0;
   S700_BT_CODE_2117.RBT1_STANDARD_WELD_DATA := W#16#0;
   S700_BT_CODE_2117.RBT2_STANDARD_WELD_DATA := W#16#0;
   S700_BT_CODE_2117.RBT3_STANDARD_WELD_DATA := W#16#0;
   S700_BT_CODE_2117.RBT4_STANDARD_WELD_DATA := W#16#0;
   S700_BT_CODE_2117.RBT5_STANDARD_WELD_DATA := W#16#0;
   S700_BT_CODE_2117.RBT6_STANDARD_WELD_DATA := W#16#0;
   S700_BT_CODE_2117.RBT7_STANDARD_WELD_DATA := W#16#0;
   S700_BT_CODE_2117.RBT8_STANDARD_WELD_DATA := W#16#0;
   S700_BT_CODE_2117.RBT9_STANDARD_WELD_DATA := W#16#0;
   S700_BT_CODE_2117.RBT10_STANDARD_WELD_DATA := W#16#0;
   S700_BT_CODE_2117.RBT11_STANDARD_WELD_DATA := W#16#0;
   S700_BT_CODE_2117.RBT12_STANDARD_WELD_DATA := W#16#0;
   S700_BT_CODE_2117.RBT13_STANDARD_WELD_DATA := W#16#0;
   S700_BT_CODE_2117.RBT14_STANDARD_WELD_DATA := W#16#0;
   S700_BT_CODE_2117.RBT15_STANDARD_WELD_DATA := W#16#0;
   S700_BT_CODE_2117.RBT16_STANDARD_WELD_DATA := W#16#0;
   S700_BT_CODE_2117.RBT17_STANDARD_WELD_DATA := W#16#0;
   S700_BT_CODE_2117.RBT18_STANDARD_WELD_DATA := W#16#0;
   S700_BT_CODE_2117.RBT19_STANDARD_WELD_DATA := W#16#0;
   S700_BT_CODE_2117.RBT20_STANDARD_WELD_DATA := W#16#0;
   S700_BT_CODE_2117.RBT21_STANDARD_WELD_DATA := W#16#0;
   S700_BT_CODE_2117.RBT22_STANDARD_WELD_DATA := W#16#0;
   S700_BT_CODE_2117.RBT23_STANDARD_WELD_DAT := W#16#0;
   S700_BT_CODE_2117.RBT24_STANDARD_WELD_DAT := W#16#0;
   S700_BT_CODE_2117.CHK_WORD := W#16#0;
   S700_BT_CODE_2117.TEST_TEMP[1] := B#16#0;
   S700_BT_CODE_2117.TEST_TEMP[2] := B#16#0;
   S700_BT_CODE_2117.TEST_TEMP[3] := B#16#0;
   S700_BT_CODE_2117.TEST_TEMP[4] := B#16#0;
   S700_BT_CODE_2117.TEST_TEMP[5] := B#16#0;
   S700_BT_CODE_2117.TEST_TEMP[6] := B#16#0;
   S700_BT_CODE_2117.TEST_TEMP[7] := B#16#0;
   S700_BT_CODE_2117.TEST_TEMP[8] := B#16#0;
   S700_BT_CODE_2117.TEST_TEMP[9] := B#16#0;
   S700_BT_CODE_2117.TEST_TEMP[10] := B#16#0;
   S700_BT_CODE_2117.TEST_TEMP[11] := B#16#0;
   S700_BT_CODE_2117.TEST_TEMP[12] := B#16#0;
   S700_BT_CODE_2117.TEST_TEMP[13] := B#16#0;
   S700_BT_CODE_2117.TEST_TEMP[14] := B#16#0;
   S700_BT_CODE_2117.TEST_TEMP[15] := B#16#0;
   S700_BT_CODE_2117.TEST_TEMP[16] := B#16#0;
   S700_BT_CODE_2117.TEST_TEMP[17] := B#16#0;
   S700_BT_CODE_2117.TEST_TEMP[18] := B#16#0;
   S700_BT_CODE_2117.TEST_TEMP[19] := B#16#0;
   S700_BT_CODE_2117.TEST_TEMP[20] := B#16#0;
   S700_BT_CODE_2117.TEST_TEMP[21] := B#16#0;
   S700_BT_CODE_2117.TEST_TEMP[22] := B#16#0;
   S700_BT_CODE_2117.TEST_TEMP[23] := B#16#0;
   S700_BT_CODE_2117.TEST_TEMP[24] := B#16#0;
   S700_BT_CODE_2117.TEST_TEMP[25] := B#16#0;
   S700_BT_CODE_2117.TEST_TEMP[26] := B#16#0;
   S700_BT_CODE_2117.TEST_TEMP[27] := B#16#0;
   S700_BT_CODE_2117.TEST_TEMP[28] := B#16#0;
   S700_BT_CODE_2117.TEST_TEMP[29] := B#16#0;
   S700_BT_CODE_2117.TEST_TEMP[30] := B#16#0;
   S700_BT_CODE_2117.TEST_TEMP[31] := B#16#0;
   S700_BT_CODE_2117.TEST_TEMP[32] := B#16#0;
   S700_BT_CODE_2117.TEST_TEMP[33] := B#16#0;
   S700_BT_CODE_2117.TEST_TEMP[34] := B#16#0;
   S700_BT_CODE_2117.TEST_TEMP[35] := B#16#0;
   S700_BT_CODE_2117.TEST_TEMP[36] := B#16#0;
   S700_BT_CODE_2117.TEST_TEMP[37] := B#16#0;
   S700_BT_CODE_2117.TEST_TEMP[38] := B#16#0;
   S700_BT_CODE_2117.TEST_TEMP[39] := B#16#0;
   S700_BT_CODE_2117.TEST_TEMP[40] := B#16#0;
   S700_BT_CODE_2118.STATION_MAIN := W#16#0;
   S700_BT_CODE_2118.DISTINCTION_LH_RH := W#16#0;
   S700_BT_CODE_2118.STAION_NUMBER := W#16#0;
   S700_BT_CODE_2118.BODY_TYPE_1ST := W#16#0;
   S700_BT_CODE_2118.BODY_TYPE_OPTION := W#16#0;
   S700_BT_CODE_2118.RBT1_STANDARD_WELD_DATA := W#16#0;
   S700_BT_CODE_2118.RBT2_STANDARD_WELD_DATA := W#16#0;
   S700_BT_CODE_2118.RBT3_STANDARD_WELD_DATA := W#16#0;
   S700_BT_CODE_2118.RBT4_STANDARD_WELD_DATA := W#16#0;
   S700_BT_CODE_2118.RBT5_STANDARD_WELD_DATA := W#16#0;
   S700_BT_CODE_2118.RBT6_STANDARD_WELD_DATA := W#16#0;
   S700_BT_CODE_2118.RBT7_STANDARD_WELD_DATA := W#16#0;
   S700_BT_CODE_2118.RBT8_STANDARD_WELD_DATA := W#16#0;
   S700_BT_CODE_2118.RBT9_STANDARD_WELD_DATA := W#16#0;
   S700_BT_CODE_2118.RBT10_STANDARD_WELD_DATA := W#16#0;
   S700_BT_CODE_2118.RBT11_STANDARD_WELD_DATA := W#16#0;
   S700_BT_CODE_2118.RBT12_STANDARD_WELD_DATA := W#16#0;
   S700_BT_CODE_2118.RBT13_STANDARD_WELD_DATA := W#16#0;
   S700_BT_CODE_2118.RBT14_STANDARD_WELD_DATA := W#16#0;
   S700_BT_CODE_2118.RBT15_STANDARD_WELD_DATA := W#16#0;
   S700_BT_CODE_2118.RBT16_STANDARD_WELD_DATA := W#16#0;
   S700_BT_CODE_2118.RBT17_STANDARD_WELD_DATA := W#16#0;
   S700_BT_CODE_2118.RBT18_STANDARD_WELD_DATA := W#16#0;
   S700_BT_CODE_2118.RBT19_STANDARD_WELD_DATA := W#16#0;
   S700_BT_CODE_2118.RBT20_STANDARD_WELD_DATA := W#16#0;
   S700_BT_CODE_2118.RBT21_STANDARD_WELD_DATA := W#16#0;
   S700_BT_CODE_2118.RBT22_STANDARD_WELD_DATA := W#16#0;
   S700_BT_CODE_2118.RBT23_STANDARD_WELD_DAT := W#16#0;
   S700_BT_CODE_2118.RBT24_STANDARD_WELD_DAT := W#16#0;
   S700_BT_CODE_2118.CHK_WORD := W#16#0;
   S700_BT_CODE_2118.TEST_TEMP[1] := B#16#0;
   S700_BT_CODE_2118.TEST_TEMP[2] := B#16#0;
   S700_BT_CODE_2118.TEST_TEMP[3] := B#16#0;
   S700_BT_CODE_2118.TEST_TEMP[4] := B#16#0;
   S700_BT_CODE_2118.TEST_TEMP[5] := B#16#0;
   S700_BT_CODE_2118.TEST_TEMP[6] := B#16#0;
   S700_BT_CODE_2118.TEST_TEMP[7] := B#16#0;
   S700_BT_CODE_2118.TEST_TEMP[8] := B#16#0;
   S700_BT_CODE_2118.TEST_TEMP[9] := B#16#0;
   S700_BT_CODE_2118.TEST_TEMP[10] := B#16#0;
   S700_BT_CODE_2118.TEST_TEMP[11] := B#16#0;
   S700_BT_CODE_2118.TEST_TEMP[12] := B#16#0;
   S700_BT_CODE_2118.TEST_TEMP[13] := B#16#0;
   S700_BT_CODE_2118.TEST_TEMP[14] := B#16#0;
   S700_BT_CODE_2118.TEST_TEMP[15] := B#16#0;
   S700_BT_CODE_2118.TEST_TEMP[16] := B#16#0;
   S700_BT_CODE_2118.TEST_TEMP[17] := B#16#0;
   S700_BT_CODE_2118.TEST_TEMP[18] := B#16#0;
   S700_BT_CODE_2118.TEST_TEMP[19] := B#16#0;
   S700_BT_CODE_2118.TEST_TEMP[20] := B#16#0;
   S700_BT_CODE_2118.TEST_TEMP[21] := B#16#0;
   S700_BT_CODE_2118.TEST_TEMP[22] := B#16#0;
   S700_BT_CODE_2118.TEST_TEMP[23] := B#16#0;
   S700_BT_CODE_2118.TEST_TEMP[24] := B#16#0;
   S700_BT_CODE_2118.TEST_TEMP[25] := B#16#0;
   S700_BT_CODE_2118.TEST_TEMP[26] := B#16#0;
   S700_BT_CODE_2118.TEST_TEMP[27] := B#16#0;
   S700_BT_CODE_2118.TEST_TEMP[28] := B#16#0;
   S700_BT_CODE_2118.TEST_TEMP[29] := B#16#0;
   S700_BT_CODE_2118.TEST_TEMP[30] := B#16#0;
   S700_BT_CODE_2118.TEST_TEMP[31] := B#16#0;
   S700_BT_CODE_2118.TEST_TEMP[32] := B#16#0;
   S700_BT_CODE_2118.TEST_TEMP[33] := B#16#0;
   S700_BT_CODE_2118.TEST_TEMP[34] := B#16#0;
   S700_BT_CODE_2118.TEST_TEMP[35] := B#16#0;
   S700_BT_CODE_2118.TEST_TEMP[36] := B#16#0;
   S700_BT_CODE_2118.TEST_TEMP[37] := B#16#0;
   S700_BT_CODE_2118.TEST_TEMP[38] := B#16#0;
   S700_BT_CODE_2118.TEST_TEMP[39] := B#16#0;
   S700_BT_CODE_2118.TEST_TEMP[40] := B#16#0;
   S700_BT_CODE_2119.STATION_MAIN := W#16#0;
   S700_BT_CODE_2119.DISTINCTION_LH_RH := W#16#0;
   S700_BT_CODE_2119.STAION_NUMBER := W#16#0;
   S700_BT_CODE_2119.BODY_TYPE_1ST := W#16#0;
   S700_BT_CODE_2119.BODY_TYPE_OPTION := W#16#0;
   S700_BT_CODE_2119.RBT1_STANDARD_WELD_DATA := W#16#0;
   S700_BT_CODE_2119.RBT2_STANDARD_WELD_DATA := W#16#0;
   S700_BT_CODE_2119.RBT3_STANDARD_WELD_DATA := W#16#0;
   S700_BT_CODE_2119.RBT4_STANDARD_WELD_DATA := W#16#0;
   S700_BT_CODE_2119.RBT5_STANDARD_WELD_DATA := W#16#0;
   S700_BT_CODE_2119.RBT6_STANDARD_WELD_DATA := W#16#0;
   S700_BT_CODE_2119.RBT7_STANDARD_WELD_DATA := W#16#0;
   S700_BT_CODE_2119.RBT8_STANDARD_WELD_DATA := W#16#0;
   S700_BT_CODE_2119.RBT9_STANDARD_WELD_DATA := W#16#0;
   S700_BT_CODE_2119.RBT10_STANDARD_WELD_DATA := W#16#0;
   S700_BT_CODE_2119.RBT11_STANDARD_WELD_DATA := W#16#0;
   S700_BT_CODE_2119.RBT12_STANDARD_WELD_DATA := W#16#0;
   S700_BT_CODE_2119.RBT13_STANDARD_WELD_DATA := W#16#0;
   S700_BT_CODE_2119.RBT14_STANDARD_WELD_DATA := W#16#0;
   S700_BT_CODE_2119.RBT15_STANDARD_WELD_DATA := W#16#0;
   S700_BT_CODE_2119.RBT16_STANDARD_WELD_DATA := W#16#0;
   S700_BT_CODE_2119.RBT17_STANDARD_WELD_DATA := W#16#0;
   S700_BT_CODE_2119.RBT18_STANDARD_WELD_DATA := W#16#0;
   S700_BT_CODE_2119.RBT19_STANDARD_WELD_DATA := W#16#0;
   S700_BT_CODE_2119.RBT20_STANDARD_WELD_DATA := W#16#0;
   S700_BT_CODE_2119.RBT21_STANDARD_WELD_DATA := W#16#0;
   S700_BT_CODE_2119.RBT22_STANDARD_WELD_DATA := W#16#0;
   S700_BT_CODE_2119.RBT23_STANDARD_WELD_DAT := W#16#0;
   S700_BT_CODE_2119.RBT24_STANDARD_WELD_DAT := W#16#0;
   S700_BT_CODE_2119.CHK_WORD := W#16#0;
   S700_BT_CODE_2119.TEST_TEMP[1] := B#16#0;
   S700_BT_CODE_2119.TEST_TEMP[2] := B#16#0;
   S700_BT_CODE_2119.TEST_TEMP[3] := B#16#0;
   S700_BT_CODE_2119.TEST_TEMP[4] := B#16#0;
   S700_BT_CODE_2119.TEST_TEMP[5] := B#16#0;
   S700_BT_CODE_2119.TEST_TEMP[6] := B#16#0;
   S700_BT_CODE_2119.TEST_TEMP[7] := B#16#0;
   S700_BT_CODE_2119.TEST_TEMP[8] := B#16#0;
   S700_BT_CODE_2119.TEST_TEMP[9] := B#16#0;
   S700_BT_CODE_2119.TEST_TEMP[10] := B#16#0;
   S700_BT_CODE_2119.TEST_TEMP[11] := B#16#0;
   S700_BT_CODE_2119.TEST_TEMP[12] := B#16#0;
   S700_BT_CODE_2119.TEST_TEMP[13] := B#16#0;
   S700_BT_CODE_2119.TEST_TEMP[14] := B#16#0;
   S700_BT_CODE_2119.TEST_TEMP[15] := B#16#0;
   S700_BT_CODE_2119.TEST_TEMP[16] := B#16#0;
   S700_BT_CODE_2119.TEST_TEMP[17] := B#16#0;
   S700_BT_CODE_2119.TEST_TEMP[18] := B#16#0;
   S700_BT_CODE_2119.TEST_TEMP[19] := B#16#0;
   S700_BT_CODE_2119.TEST_TEMP[20] := B#16#0;
   S700_BT_CODE_2119.TEST_TEMP[21] := B#16#0;
   S700_BT_CODE_2119.TEST_TEMP[22] := B#16#0;
   S700_BT_CODE_2119.TEST_TEMP[23] := B#16#0;
   S700_BT_CODE_2119.TEST_TEMP[24] := B#16#0;
   S700_BT_CODE_2119.TEST_TEMP[25] := B#16#0;
   S700_BT_CODE_2119.TEST_TEMP[26] := B#16#0;
   S700_BT_CODE_2119.TEST_TEMP[27] := B#16#0;
   S700_BT_CODE_2119.TEST_TEMP[28] := B#16#0;
   S700_BT_CODE_2119.TEST_TEMP[29] := B#16#0;
   S700_BT_CODE_2119.TEST_TEMP[30] := B#16#0;
   S700_BT_CODE_2119.TEST_TEMP[31] := B#16#0;
   S700_BT_CODE_2119.TEST_TEMP[32] := B#16#0;
   S700_BT_CODE_2119.TEST_TEMP[33] := B#16#0;
   S700_BT_CODE_2119.TEST_TEMP[34] := B#16#0;
   S700_BT_CODE_2119.TEST_TEMP[35] := B#16#0;
   S700_BT_CODE_2119.TEST_TEMP[36] := B#16#0;
   S700_BT_CODE_2119.TEST_TEMP[37] := B#16#0;
   S700_BT_CODE_2119.TEST_TEMP[38] := B#16#0;
   S700_BT_CODE_2119.TEST_TEMP[39] := B#16#0;
   S700_BT_CODE_2119.TEST_TEMP[40] := B#16#0;
   S700_BT_CODE_2120.STATION_MAIN := W#16#0;
   S700_BT_CODE_2120.DISTINCTION_LH_RH := W#16#0;
   S700_BT_CODE_2120.STAION_NUMBER := W#16#0;
   S700_BT_CODE_2120.BODY_TYPE_1ST := W#16#0;
   S700_BT_CODE_2120.BODY_TYPE_OPTION := W#16#0;
   S700_BT_CODE_2120.RBT1_STANDARD_WELD_DATA := W#16#0;
   S700_BT_CODE_2120.RBT2_STANDARD_WELD_DATA := W#16#0;
   S700_BT_CODE_2120.RBT3_STANDARD_WELD_DATA := W#16#0;
   S700_BT_CODE_2120.RBT4_STANDARD_WELD_DATA := W#16#0;
   S700_BT_CODE_2120.RBT5_STANDARD_WELD_DATA := W#16#0;
   S700_BT_CODE_2120.RBT6_STANDARD_WELD_DATA := W#16#0;
   S700_BT_CODE_2120.RBT7_STANDARD_WELD_DATA := W#16#0;
   S700_BT_CODE_2120.RBT8_STANDARD_WELD_DATA := W#16#0;
   S700_BT_CODE_2120.RBT9_STANDARD_WELD_DATA := W#16#0;
   S700_BT_CODE_2120.RBT10_STANDARD_WELD_DATA := W#16#0;
   S700_BT_CODE_2120.RBT11_STANDARD_WELD_DATA := W#16#0;
   S700_BT_CODE_2120.RBT12_STANDARD_WELD_DATA := W#16#0;
   S700_BT_CODE_2120.RBT13_STANDARD_WELD_DATA := W#16#0;
   S700_BT_CODE_2120.RBT14_STANDARD_WELD_DATA := W#16#0;
   S700_BT_CODE_2120.RBT15_STANDARD_WELD_DATA := W#16#0;
   S700_BT_CODE_2120.RBT16_STANDARD_WELD_DATA := W#16#0;
   S700_BT_CODE_2120.RBT17_STANDARD_WELD_DATA := W#16#0;
   S700_BT_CODE_2120.RBT18_STANDARD_WELD_DATA := W#16#0;
   S700_BT_CODE_2120.RBT19_STANDARD_WELD_DATA := W#16#0;
   S700_BT_CODE_2120.RBT20_STANDARD_WELD_DATA := W#16#0;
   S700_BT_CODE_2120.RBT21_STANDARD_WELD_DATA := W#16#0;
   S700_BT_CODE_2120.RBT22_STANDARD_WELD_DATA := W#16#0;
   S700_BT_CODE_2120.RBT23_STANDARD_WELD_DAT := W#16#0;
   S700_BT_CODE_2120.RBT24_STANDARD_WELD_DAT := W#16#0;
   S700_BT_CODE_2120.CHK_WORD := W#16#0;
   S700_BT_CODE_2120.TEST_TEMP[1] := B#16#0;
   S700_BT_CODE_2120.TEST_TEMP[2] := B#16#0;
   S700_BT_CODE_2120.TEST_TEMP[3] := B#16#0;
   S700_BT_CODE_2120.TEST_TEMP[4] := B#16#0;
   S700_BT_CODE_2120.TEST_TEMP[5] := B#16#0;
   S700_BT_CODE_2120.TEST_TEMP[6] := B#16#0;
   S700_BT_CODE_2120.TEST_TEMP[7] := B#16#0;
   S700_BT_CODE_2120.TEST_TEMP[8] := B#16#0;
   S700_BT_CODE_2120.TEST_TEMP[9] := B#16#0;
   S700_BT_CODE_2120.TEST_TEMP[10] := B#16#0;
   S700_BT_CODE_2120.TEST_TEMP[11] := B#16#0;
   S700_BT_CODE_2120.TEST_TEMP[12] := B#16#0;
   S700_BT_CODE_2120.TEST_TEMP[13] := B#16#0;
   S700_BT_CODE_2120.TEST_TEMP[14] := B#16#0;
   S700_BT_CODE_2120.TEST_TEMP[15] := B#16#0;
   S700_BT_CODE_2120.TEST_TEMP[16] := B#16#0;
   S700_BT_CODE_2120.TEST_TEMP[17] := B#16#0;
   S700_BT_CODE_2120.TEST_TEMP[18] := B#16#0;
   S700_BT_CODE_2120.TEST_TEMP[19] := B#16#0;
   S700_BT_CODE_2120.TEST_TEMP[20] := B#16#0;
   S700_BT_CODE_2120.TEST_TEMP[21] := B#16#0;
   S700_BT_CODE_2120.TEST_TEMP[22] := B#16#0;
   S700_BT_CODE_2120.TEST_TEMP[23] := B#16#0;
   S700_BT_CODE_2120.TEST_TEMP[24] := B#16#0;
   S700_BT_CODE_2120.TEST_TEMP[25] := B#16#0;
   S700_BT_CODE_2120.TEST_TEMP[26] := B#16#0;
   S700_BT_CODE_2120.TEST_TEMP[27] := B#16#0;
   S700_BT_CODE_2120.TEST_TEMP[28] := B#16#0;
   S700_BT_CODE_2120.TEST_TEMP[29] := B#16#0;
   S700_BT_CODE_2120.TEST_TEMP[30] := B#16#0;
   S700_BT_CODE_2120.TEST_TEMP[31] := B#16#0;
   S700_BT_CODE_2120.TEST_TEMP[32] := B#16#0;
   S700_BT_CODE_2120.TEST_TEMP[33] := B#16#0;
   S700_BT_CODE_2120.TEST_TEMP[34] := B#16#0;
   S700_BT_CODE_2120.TEST_TEMP[35] := B#16#0;
   S700_BT_CODE_2120.TEST_TEMP[36] := B#16#0;
   S700_BT_CODE_2120.TEST_TEMP[37] := B#16#0;
   S700_BT_CODE_2120.TEST_TEMP[38] := B#16#0;
   S700_BT_CODE_2120.TEST_TEMP[39] := B#16#0;
   S700_BT_CODE_2120.TEST_TEMP[40] := B#16#0;
   S700_1_BT_CODE_2101.STATION_MAIN := W#16#0;
   S700_1_BT_CODE_2101.DISTINCTION_LH_RH := W#16#0;
   S700_1_BT_CODE_2101.STAION_NUMBER := W#16#0;
   S700_1_BT_CODE_2101.BODY_TYPE_1ST := W#16#0;
   S700_1_BT_CODE_2101.BODY_TYPE_OPTION := W#16#0;
   S700_1_BT_CODE_2101.RBT1_STANDARD_WELD_DATA := W#16#0;
   S700_1_BT_CODE_2101.RBT2_STANDARD_WELD_DATA := W#16#0;
   S700_1_BT_CODE_2101.RBT3_STANDARD_WELD_DATA := W#16#0;
   S700_1_BT_CODE_2101.RBT4_STANDARD_WELD_DATA := W#16#0;
   S700_1_BT_CODE_2101.RBT5_STANDARD_WELD_DATA := W#16#0;
   S700_1_BT_CODE_2101.RBT6_STANDARD_WELD_DATA := W#16#0;
   S700_1_BT_CODE_2101.RBT7_STANDARD_WELD_DATA := W#16#0;
   S700_1_BT_CODE_2101.RBT8_STANDARD_WELD_DATA := W#16#0;
   S700_1_BT_CODE_2101.RBT9_STANDARD_WELD_DATA := W#16#0;
   S700_1_BT_CODE_2101.RBT10_STANDARD_WELD_DATA := W#16#0;
   S700_1_BT_CODE_2101.RBT11_STANDARD_WELD_DATA := W#16#0;
   S700_1_BT_CODE_2101.RBT12_STANDARD_WELD_DATA := W#16#0;
   S700_1_BT_CODE_2101.RBT13_STANDARD_WELD_DATA := W#16#0;
   S700_1_BT_CODE_2101.RBT14_STANDARD_WELD_DATA := W#16#0;
   S700_1_BT_CODE_2101.RBT15_STANDARD_WELD_DATA := W#16#0;
   S700_1_BT_CODE_2101.RBT16_STANDARD_WELD_DATA := W#16#0;
   S700_1_BT_CODE_2101.RBT17_STANDARD_WELD_DATA := W#16#0;
   S700_1_BT_CODE_2101.RBT18_STANDARD_WELD_DATA := W#16#0;
   S700_1_BT_CODE_2101.RBT19_STANDARD_WELD_DATA := W#16#0;
   S700_1_BT_CODE_2101.RBT20_STANDARD_WELD_DATA := W#16#0;
   S700_1_BT_CODE_2101.RBT21_STANDARD_WELD_DATA := W#16#0;
   S700_1_BT_CODE_2101.RBT22_STANDARD_WELD_DATA := W#16#0;
   S700_1_BT_CODE_2101.RBT23_STANDARD_WELD_DAT := W#16#0;
   S700_1_BT_CODE_2101.RBT24_STANDARD_WELD_DAT := W#16#0;
   S700_1_BT_CODE_2101.CHK_WORD := W#16#0;
   S700_1_BT_CODE_2101.TEST_TEMP[1] := B#16#0;
   S700_1_BT_CODE_2101.TEST_TEMP[2] := B#16#0;
   S700_1_BT_CODE_2101.TEST_TEMP[3] := B#16#0;
   S700_1_BT_CODE_2101.TEST_TEMP[4] := B#16#0;
   S700_1_BT_CODE_2101.TEST_TEMP[5] := B#16#0;
   S700_1_BT_CODE_2101.TEST_TEMP[6] := B#16#0;
   S700_1_BT_CODE_2101.TEST_TEMP[7] := B#16#0;
   S700_1_BT_CODE_2101.TEST_TEMP[8] := B#16#0;
   S700_1_BT_CODE_2101.TEST_TEMP[9] := B#16#0;
   S700_1_BT_CODE_2101.TEST_TEMP[10] := B#16#0;
   S700_1_BT_CODE_2101.TEST_TEMP[11] := B#16#0;
   S700_1_BT_CODE_2101.TEST_TEMP[12] := B#16#0;
   S700_1_BT_CODE_2101.TEST_TEMP[13] := B#16#0;
   S700_1_BT_CODE_2101.TEST_TEMP[14] := B#16#0;
   S700_1_BT_CODE_2101.TEST_TEMP[15] := B#16#0;
   S700_1_BT_CODE_2101.TEST_TEMP[16] := B#16#0;
   S700_1_BT_CODE_2101.TEST_TEMP[17] := B#16#0;
   S700_1_BT_CODE_2101.TEST_TEMP[18] := B#16#0;
   S700_1_BT_CODE_2101.TEST_TEMP[19] := B#16#0;
   S700_1_BT_CODE_2101.TEST_TEMP[20] := B#16#0;
   S700_1_BT_CODE_2101.TEST_TEMP[21] := B#16#0;
   S700_1_BT_CODE_2101.TEST_TEMP[22] := B#16#0;
   S700_1_BT_CODE_2101.TEST_TEMP[23] := B#16#0;
   S700_1_BT_CODE_2101.TEST_TEMP[24] := B#16#0;
   S700_1_BT_CODE_2101.TEST_TEMP[25] := B#16#0;
   S700_1_BT_CODE_2101.TEST_TEMP[26] := B#16#0;
   S700_1_BT_CODE_2101.TEST_TEMP[27] := B#16#0;
   S700_1_BT_CODE_2101.TEST_TEMP[28] := B#16#0;
   S700_1_BT_CODE_2101.TEST_TEMP[29] := B#16#0;
   S700_1_BT_CODE_2101.TEST_TEMP[30] := B#16#0;
   S700_1_BT_CODE_2101.TEST_TEMP[31] := B#16#0;
   S700_1_BT_CODE_2101.TEST_TEMP[32] := B#16#0;
   S700_1_BT_CODE_2101.TEST_TEMP[33] := B#16#0;
   S700_1_BT_CODE_2101.TEST_TEMP[34] := B#16#0;
   S700_1_BT_CODE_2101.TEST_TEMP[35] := B#16#0;
   S700_1_BT_CODE_2101.TEST_TEMP[36] := B#16#0;
   S700_1_BT_CODE_2101.TEST_TEMP[37] := B#16#0;
   S700_1_BT_CODE_2101.TEST_TEMP[38] := B#16#0;
   S700_1_BT_CODE_2101.TEST_TEMP[39] := B#16#0;
   S700_1_BT_CODE_2101.TEST_TEMP[40] := B#16#0;
   S700_1_BT_CODE_2102.STATION_MAIN := W#16#0;
   S700_1_BT_CODE_2102.DISTINCTION_LH_RH := W#16#0;
   S700_1_BT_CODE_2102.STAION_NUMBER := W#16#0;
   S700_1_BT_CODE_2102.BODY_TYPE_1ST := W#16#0;
   S700_1_BT_CODE_2102.BODY_TYPE_OPTION := W#16#0;
   S700_1_BT_CODE_2102.RBT1_STANDARD_WELD_DATA := W#16#0;
   S700_1_BT_CODE_2102.RBT2_STANDARD_WELD_DATA := W#16#0;
   S700_1_BT_CODE_2102.RBT3_STANDARD_WELD_DATA := W#16#0;
   S700_1_BT_CODE_2102.RBT4_STANDARD_WELD_DATA := W#16#0;
   S700_1_BT_CODE_2102.RBT5_STANDARD_WELD_DATA := W#16#0;
   S700_1_BT_CODE_2102.RBT6_STANDARD_WELD_DATA := W#16#0;
   S700_1_BT_CODE_2102.RBT7_STANDARD_WELD_DATA := W#16#0;
   S700_1_BT_CODE_2102.RBT8_STANDARD_WELD_DATA := W#16#0;
   S700_1_BT_CODE_2102.RBT9_STANDARD_WELD_DATA := W#16#0;
   S700_1_BT_CODE_2102.RBT10_STANDARD_WELD_DATA := W#16#0;
   S700_1_BT_CODE_2102.RBT11_STANDARD_WELD_DATA := W#16#0;
   S700_1_BT_CODE_2102.RBT12_STANDARD_WELD_DATA := W#16#0;
   S700_1_BT_CODE_2102.RBT13_STANDARD_WELD_DATA := W#16#0;
   S700_1_BT_CODE_2102.RBT14_STANDARD_WELD_DATA := W#16#0;
   S700_1_BT_CODE_2102.RBT15_STANDARD_WELD_DATA := W#16#0;
   S700_1_BT_CODE_2102.RBT16_STANDARD_WELD_DATA := W#16#0;
   S700_1_BT_CODE_2102.RBT17_STANDARD_WELD_DATA := W#16#0;
   S700_1_BT_CODE_2102.RBT18_STANDARD_WELD_DATA := W#16#0;
   S700_1_BT_CODE_2102.RBT19_STANDARD_WELD_DATA := W#16#0;
   S700_1_BT_CODE_2102.RBT20_STANDARD_WELD_DATA := W#16#0;
   S700_1_BT_CODE_2102.RBT21_STANDARD_WELD_DATA := W#16#0;
   S700_1_BT_CODE_2102.RBT22_STANDARD_WELD_DATA := W#16#0;
   S700_1_BT_CODE_2102.RBT23_STANDARD_WELD_DAT := W#16#0;
   S700_1_BT_CODE_2102.RBT24_STANDARD_WELD_DAT := W#16#0;
   S700_1_BT_CODE_2102.CHK_WORD := W#16#0;
   S700_1_BT_CODE_2102.TEST_TEMP[1] := B#16#0;
   S700_1_BT_CODE_2102.TEST_TEMP[2] := B#16#0;
   S700_1_BT_CODE_2102.TEST_TEMP[3] := B#16#0;
   S700_1_BT_CODE_2102.TEST_TEMP[4] := B#16#0;
   S700_1_BT_CODE_2102.TEST_TEMP[5] := B#16#0;
   S700_1_BT_CODE_2102.TEST_TEMP[6] := B#16#0;
   S700_1_BT_CODE_2102.TEST_TEMP[7] := B#16#0;
   S700_1_BT_CODE_2102.TEST_TEMP[8] := B#16#0;
   S700_1_BT_CODE_2102.TEST_TEMP[9] := B#16#0;
   S700_1_BT_CODE_2102.TEST_TEMP[10] := B#16#0;
   S700_1_BT_CODE_2102.TEST_TEMP[11] := B#16#0;
   S700_1_BT_CODE_2102.TEST_TEMP[12] := B#16#0;
   S700_1_BT_CODE_2102.TEST_TEMP[13] := B#16#0;
   S700_1_BT_CODE_2102.TEST_TEMP[14] := B#16#0;
   S700_1_BT_CODE_2102.TEST_TEMP[15] := B#16#0;
   S700_1_BT_CODE_2102.TEST_TEMP[16] := B#16#0;
   S700_1_BT_CODE_2102.TEST_TEMP[17] := B#16#0;
   S700_1_BT_CODE_2102.TEST_TEMP[18] := B#16#0;
   S700_1_BT_CODE_2102.TEST_TEMP[19] := B#16#0;
   S700_1_BT_CODE_2102.TEST_TEMP[20] := B#16#0;
   S700_1_BT_CODE_2102.TEST_TEMP[21] := B#16#0;
   S700_1_BT_CODE_2102.TEST_TEMP[22] := B#16#0;
   S700_1_BT_CODE_2102.TEST_TEMP[23] := B#16#0;
   S700_1_BT_CODE_2102.TEST_TEMP[24] := B#16#0;
   S700_1_BT_CODE_2102.TEST_TEMP[25] := B#16#0;
   S700_1_BT_CODE_2102.TEST_TEMP[26] := B#16#0;
   S700_1_BT_CODE_2102.TEST_TEMP[27] := B#16#0;
   S700_1_BT_CODE_2102.TEST_TEMP[28] := B#16#0;
   S700_1_BT_CODE_2102.TEST_TEMP[29] := B#16#0;
   S700_1_BT_CODE_2102.TEST_TEMP[30] := B#16#0;
   S700_1_BT_CODE_2102.TEST_TEMP[31] := B#16#0;
   S700_1_BT_CODE_2102.TEST_TEMP[32] := B#16#0;
   S700_1_BT_CODE_2102.TEST_TEMP[33] := B#16#0;
   S700_1_BT_CODE_2102.TEST_TEMP[34] := B#16#0;
   S700_1_BT_CODE_2102.TEST_TEMP[35] := B#16#0;
   S700_1_BT_CODE_2102.TEST_TEMP[36] := B#16#0;
   S700_1_BT_CODE_2102.TEST_TEMP[37] := B#16#0;
   S700_1_BT_CODE_2102.TEST_TEMP[38] := B#16#0;
   S700_1_BT_CODE_2102.TEST_TEMP[39] := B#16#0;
   S700_1_BT_CODE_2102.TEST_TEMP[40] := B#16#0;
   S700_1_BT_CODE_2103.STATION_MAIN := W#16#0;
   S700_1_BT_CODE_2103.DISTINCTION_LH_RH := W#16#0;
   S700_1_BT_CODE_2103.STAION_NUMBER := W#16#0;
   S700_1_BT_CODE_2103.BODY_TYPE_1ST := W#16#0;
   S700_1_BT_CODE_2103.BODY_TYPE_OPTION := W#16#0;
   S700_1_BT_CODE_2103.RBT1_STANDARD_WELD_DATA := W#16#0;
   S700_1_BT_CODE_2103.RBT2_STANDARD_WELD_DATA := W#16#0;
   S700_1_BT_CODE_2103.RBT3_STANDARD_WELD_DATA := W#16#0;
   S700_1_BT_CODE_2103.RBT4_STANDARD_WELD_DATA := W#16#0;
   S700_1_BT_CODE_2103.RBT5_STANDARD_WELD_DATA := W#16#0;
   S700_1_BT_CODE_2103.RBT6_STANDARD_WELD_DATA := W#16#0;
   S700_1_BT_CODE_2103.RBT7_STANDARD_WELD_DATA := W#16#0;
   S700_1_BT_CODE_2103.RBT8_STANDARD_WELD_DATA := W#16#0;
   S700_1_BT_CODE_2103.RBT9_STANDARD_WELD_DATA := W#16#0;
   S700_1_BT_CODE_2103.RBT10_STANDARD_WELD_DATA := W#16#0;
   S700_1_BT_CODE_2103.RBT11_STANDARD_WELD_DATA := W#16#0;
   S700_1_BT_CODE_2103.RBT12_STANDARD_WELD_DATA := W#16#0;
   S700_1_BT_CODE_2103.RBT13_STANDARD_WELD_DATA := W#16#0;
   S700_1_BT_CODE_2103.RBT14_STANDARD_WELD_DATA := W#16#0;
   S700_1_BT_CODE_2103.RBT15_STANDARD_WELD_DATA := W#16#0;
   S700_1_BT_CODE_2103.RBT16_STANDARD_WELD_DATA := W#16#0;
   S700_1_BT_CODE_2103.RBT17_STANDARD_WELD_DATA := W#16#0;
   S700_1_BT_CODE_2103.RBT18_STANDARD_WELD_DATA := W#16#0;
   S700_1_BT_CODE_2103.RBT19_STANDARD_WELD_DATA := W#16#0;
   S700_1_BT_CODE_2103.RBT20_STANDARD_WELD_DATA := W#16#0;
   S700_1_BT_CODE_2103.RBT21_STANDARD_WELD_DATA := W#16#0;
   S700_1_BT_CODE_2103.RBT22_STANDARD_WELD_DATA := W#16#0;
   S700_1_BT_CODE_2103.RBT23_STANDARD_WELD_DAT := W#16#0;
   S700_1_BT_CODE_2103.RBT24_STANDARD_WELD_DAT := W#16#0;
   S700_1_BT_CODE_2103.CHK_WORD := W#16#0;
   S700_1_BT_CODE_2103.TEST_TEMP[1] := B#16#0;
   S700_1_BT_CODE_2103.TEST_TEMP[2] := B#16#0;
   S700_1_BT_CODE_2103.TEST_TEMP[3] := B#16#0;
   S700_1_BT_CODE_2103.TEST_TEMP[4] := B#16#0;
   S700_1_BT_CODE_2103.TEST_TEMP[5] := B#16#0;
   S700_1_BT_CODE_2103.TEST_TEMP[6] := B#16#0;
   S700_1_BT_CODE_2103.TEST_TEMP[7] := B#16#0;
   S700_1_BT_CODE_2103.TEST_TEMP[8] := B#16#0;
   S700_1_BT_CODE_2103.TEST_TEMP[9] := B#16#0;
   S700_1_BT_CODE_2103.TEST_TEMP[10] := B#16#0;
   S700_1_BT_CODE_2103.TEST_TEMP[11] := B#16#0;
   S700_1_BT_CODE_2103.TEST_TEMP[12] := B#16#0;
   S700_1_BT_CODE_2103.TEST_TEMP[13] := B#16#0;
   S700_1_BT_CODE_2103.TEST_TEMP[14] := B#16#0;
   S700_1_BT_CODE_2103.TEST_TEMP[15] := B#16#0;
   S700_1_BT_CODE_2103.TEST_TEMP[16] := B#16#0;
   S700_1_BT_CODE_2103.TEST_TEMP[17] := B#16#0;
   S700_1_BT_CODE_2103.TEST_TEMP[18] := B#16#0;
   S700_1_BT_CODE_2103.TEST_TEMP[19] := B#16#0;
   S700_1_BT_CODE_2103.TEST_TEMP[20] := B#16#0;
   S700_1_BT_CODE_2103.TEST_TEMP[21] := B#16#0;
   S700_1_BT_CODE_2103.TEST_TEMP[22] := B#16#0;
   S700_1_BT_CODE_2103.TEST_TEMP[23] := B#16#0;
   S700_1_BT_CODE_2103.TEST_TEMP[24] := B#16#0;
   S700_1_BT_CODE_2103.TEST_TEMP[25] := B#16#0;
   S700_1_BT_CODE_2103.TEST_TEMP[26] := B#16#0;
   S700_1_BT_CODE_2103.TEST_TEMP[27] := B#16#0;
   S700_1_BT_CODE_2103.TEST_TEMP[28] := B#16#0;
   S700_1_BT_CODE_2103.TEST_TEMP[29] := B#16#0;
   S700_1_BT_CODE_2103.TEST_TEMP[30] := B#16#0;
   S700_1_BT_CODE_2103.TEST_TEMP[31] := B#16#0;
   S700_1_BT_CODE_2103.TEST_TEMP[32] := B#16#0;
   S700_1_BT_CODE_2103.TEST_TEMP[33] := B#16#0;
   S700_1_BT_CODE_2103.TEST_TEMP[34] := B#16#0;
   S700_1_BT_CODE_2103.TEST_TEMP[35] := B#16#0;
   S700_1_BT_CODE_2103.TEST_TEMP[36] := B#16#0;
   S700_1_BT_CODE_2103.TEST_TEMP[37] := B#16#0;
   S700_1_BT_CODE_2103.TEST_TEMP[38] := B#16#0;
   S700_1_BT_CODE_2103.TEST_TEMP[39] := B#16#0;
   S700_1_BT_CODE_2103.TEST_TEMP[40] := B#16#0;
   S700_1_BT_CODE_2104.STATION_MAIN := W#16#0;
   S700_1_BT_CODE_2104.DISTINCTION_LH_RH := W#16#0;
   S700_1_BT_CODE_2104.STAION_NUMBER := W#16#0;
   S700_1_BT_CODE_2104.BODY_TYPE_1ST := W#16#0;
   S700_1_BT_CODE_2104.BODY_TYPE_OPTION := W#16#0;
   S700_1_BT_CODE_2104.RBT1_STANDARD_WELD_DATA := W#16#0;
   S700_1_BT_CODE_2104.RBT2_STANDARD_WELD_DATA := W#16#0;
   S700_1_BT_CODE_2104.RBT3_STANDARD_WELD_DATA := W#16#0;
   S700_1_BT_CODE_2104.RBT4_STANDARD_WELD_DATA := W#16#0;
   S700_1_BT_CODE_2104.RBT5_STANDARD_WELD_DATA := W#16#0;
   S700_1_BT_CODE_2104.RBT6_STANDARD_WELD_DATA := W#16#0;
   S700_1_BT_CODE_2104.RBT7_STANDARD_WELD_DATA := W#16#0;
   S700_1_BT_CODE_2104.RBT8_STANDARD_WELD_DATA := W#16#0;
   S700_1_BT_CODE_2104.RBT9_STANDARD_WELD_DATA := W#16#0;
   S700_1_BT_CODE_2104.RBT10_STANDARD_WELD_DATA := W#16#0;
   S700_1_BT_CODE_2104.RBT11_STANDARD_WELD_DATA := W#16#0;
   S700_1_BT_CODE_2104.RBT12_STANDARD_WELD_DATA := W#16#0;
   S700_1_BT_CODE_2104.RBT13_STANDARD_WELD_DATA := W#16#0;
   S700_1_BT_CODE_2104.RBT14_STANDARD_WELD_DATA := W#16#0;
   S700_1_BT_CODE_2104.RBT15_STANDARD_WELD_DATA := W#16#0;
   S700_1_BT_CODE_2104.RBT16_STANDARD_WELD_DATA := W#16#0;
   S700_1_BT_CODE_2104.RBT17_STANDARD_WELD_DATA := W#16#0;
   S700_1_BT_CODE_2104.RBT18_STANDARD_WELD_DATA := W#16#0;
   S700_1_BT_CODE_2104.RBT19_STANDARD_WELD_DATA := W#16#0;
   S700_1_BT_CODE_2104.RBT20_STANDARD_WELD_DATA := W#16#0;
   S700_1_BT_CODE_2104.RBT21_STANDARD_WELD_DATA := W#16#0;
   S700_1_BT_CODE_2104.RBT22_STANDARD_WELD_DATA := W#16#0;
   S700_1_BT_CODE_2104.RBT23_STANDARD_WELD_DAT := W#16#0;
   S700_1_BT_CODE_2104.RBT24_STANDARD_WELD_DAT := W#16#0;
   S700_1_BT_CODE_2104.CHK_WORD := W#16#0;
   S700_1_BT_CODE_2104.TEST_TEMP[1] := B#16#0;
   S700_1_BT_CODE_2104.TEST_TEMP[2] := B#16#0;
   S700_1_BT_CODE_2104.TEST_TEMP[3] := B#16#0;
   S700_1_BT_CODE_2104.TEST_TEMP[4] := B#16#0;
   S700_1_BT_CODE_2104.TEST_TEMP[5] := B#16#0;
   S700_1_BT_CODE_2104.TEST_TEMP[6] := B#16#0;
   S700_1_BT_CODE_2104.TEST_TEMP[7] := B#16#0;
   S700_1_BT_CODE_2104.TEST_TEMP[8] := B#16#0;
   S700_1_BT_CODE_2104.TEST_TEMP[9] := B#16#0;
   S700_1_BT_CODE_2104.TEST_TEMP[10] := B#16#0;
   S700_1_BT_CODE_2104.TEST_TEMP[11] := B#16#0;
   S700_1_BT_CODE_2104.TEST_TEMP[12] := B#16#0;
   S700_1_BT_CODE_2104.TEST_TEMP[13] := B#16#0;
   S700_1_BT_CODE_2104.TEST_TEMP[14] := B#16#0;
   S700_1_BT_CODE_2104.TEST_TEMP[15] := B#16#0;
   S700_1_BT_CODE_2104.TEST_TEMP[16] := B#16#0;
   S700_1_BT_CODE_2104.TEST_TEMP[17] := B#16#0;
   S700_1_BT_CODE_2104.TEST_TEMP[18] := B#16#0;
   S700_1_BT_CODE_2104.TEST_TEMP[19] := B#16#0;
   S700_1_BT_CODE_2104.TEST_TEMP[20] := B#16#0;
   S700_1_BT_CODE_2104.TEST_TEMP[21] := B#16#0;
   S700_1_BT_CODE_2104.TEST_TEMP[22] := B#16#0;
   S700_1_BT_CODE_2104.TEST_TEMP[23] := B#16#0;
   S700_1_BT_CODE_2104.TEST_TEMP[24] := B#16#0;
   S700_1_BT_CODE_2104.TEST_TEMP[25] := B#16#0;
   S700_1_BT_CODE_2104.TEST_TEMP[26] := B#16#0;
   S700_1_BT_CODE_2104.TEST_TEMP[27] := B#16#0;
   S700_1_BT_CODE_2104.TEST_TEMP[28] := B#16#0;
   S700_1_BT_CODE_2104.TEST_TEMP[29] := B#16#0;
   S700_1_BT_CODE_2104.TEST_TEMP[30] := B#16#0;
   S700_1_BT_CODE_2104.TEST_TEMP[31] := B#16#0;
   S700_1_BT_CODE_2104.TEST_TEMP[32] := B#16#0;
   S700_1_BT_CODE_2104.TEST_TEMP[33] := B#16#0;
   S700_1_BT_CODE_2104.TEST_TEMP[34] := B#16#0;
   S700_1_BT_CODE_2104.TEST_TEMP[35] := B#16#0;
   S700_1_BT_CODE_2104.TEST_TEMP[36] := B#16#0;
   S700_1_BT_CODE_2104.TEST_TEMP[37] := B#16#0;
   S700_1_BT_CODE_2104.TEST_TEMP[38] := B#16#0;
   S700_1_BT_CODE_2104.TEST_TEMP[39] := B#16#0;
   S700_1_BT_CODE_2104.TEST_TEMP[40] := B#16#0;
   S700_1_BT_CODE_2105.STATION_MAIN := W#16#0;
   S700_1_BT_CODE_2105.DISTINCTION_LH_RH := W#16#0;
   S700_1_BT_CODE_2105.STAION_NUMBER := W#16#0;
   S700_1_BT_CODE_2105.BODY_TYPE_1ST := W#16#0;
   S700_1_BT_CODE_2105.BODY_TYPE_OPTION := W#16#0;
   S700_1_BT_CODE_2105.RBT1_STANDARD_WELD_DATA := W#16#0;
   S700_1_BT_CODE_2105.RBT2_STANDARD_WELD_DATA := W#16#0;
   S700_1_BT_CODE_2105.RBT3_STANDARD_WELD_DATA := W#16#0;
   S700_1_BT_CODE_2105.RBT4_STANDARD_WELD_DATA := W#16#0;
   S700_1_BT_CODE_2105.RBT5_STANDARD_WELD_DATA := W#16#0;
   S700_1_BT_CODE_2105.RBT6_STANDARD_WELD_DATA := W#16#0;
   S700_1_BT_CODE_2105.RBT7_STANDARD_WELD_DATA := W#16#0;
   S700_1_BT_CODE_2105.RBT8_STANDARD_WELD_DATA := W#16#0;
   S700_1_BT_CODE_2105.RBT9_STANDARD_WELD_DATA := W#16#0;
   S700_1_BT_CODE_2105.RBT10_STANDARD_WELD_DATA := W#16#0;
   S700_1_BT_CODE_2105.RBT11_STANDARD_WELD_DATA := W#16#0;
   S700_1_BT_CODE_2105.RBT12_STANDARD_WELD_DATA := W#16#0;
   S700_1_BT_CODE_2105.RBT13_STANDARD_WELD_DATA := W#16#0;
   S700_1_BT_CODE_2105.RBT14_STANDARD_WELD_DATA := W#16#0;
   S700_1_BT_CODE_2105.RBT15_STANDARD_WELD_DATA := W#16#0;
   S700_1_BT_CODE_2105.RBT16_STANDARD_WELD_DATA := W#16#0;
   S700_1_BT_CODE_2105.RBT17_STANDARD_WELD_DATA := W#16#0;
   S700_1_BT_CODE_2105.RBT18_STANDARD_WELD_DATA := W#16#0;
   S700_1_BT_CODE_2105.RBT19_STANDARD_WELD_DATA := W#16#0;
   S700_1_BT_CODE_2105.RBT20_STANDARD_WELD_DATA := W#16#0;
   S700_1_BT_CODE_2105.RBT21_STANDARD_WELD_DATA := W#16#0;
   S700_1_BT_CODE_2105.RBT22_STANDARD_WELD_DATA := W#16#0;
   S700_1_BT_CODE_2105.RBT23_STANDARD_WELD_DAT := W#16#0;
   S700_1_BT_CODE_2105.RBT24_STANDARD_WELD_DAT := W#16#0;
   S700_1_BT_CODE_2105.CHK_WORD := W#16#0;
   S700_1_BT_CODE_2105.TEST_TEMP[1] := B#16#0;
   S700_1_BT_CODE_2105.TEST_TEMP[2] := B#16#0;
   S700_1_BT_CODE_2105.TEST_TEMP[3] := B#16#0;
   S700_1_BT_CODE_2105.TEST_TEMP[4] := B#16#0;
   S700_1_BT_CODE_2105.TEST_TEMP[5] := B#16#0;
   S700_1_BT_CODE_2105.TEST_TEMP[6] := B#16#0;
   S700_1_BT_CODE_2105.TEST_TEMP[7] := B#16#0;
   S700_1_BT_CODE_2105.TEST_TEMP[8] := B#16#0;
   S700_1_BT_CODE_2105.TEST_TEMP[9] := B#16#0;
   S700_1_BT_CODE_2105.TEST_TEMP[10] := B#16#0;
   S700_1_BT_CODE_2105.TEST_TEMP[11] := B#16#0;
   S700_1_BT_CODE_2105.TEST_TEMP[12] := B#16#0;
   S700_1_BT_CODE_2105.TEST_TEMP[13] := B#16#0;
   S700_1_BT_CODE_2105.TEST_TEMP[14] := B#16#0;
   S700_1_BT_CODE_2105.TEST_TEMP[15] := B#16#0;
   S700_1_BT_CODE_2105.TEST_TEMP[16] := B#16#0;
   S700_1_BT_CODE_2105.TEST_TEMP[17] := B#16#0;
   S700_1_BT_CODE_2105.TEST_TEMP[18] := B#16#0;
   S700_1_BT_CODE_2105.TEST_TEMP[19] := B#16#0;
   S700_1_BT_CODE_2105.TEST_TEMP[20] := B#16#0;
   S700_1_BT_CODE_2105.TEST_TEMP[21] := B#16#0;
   S700_1_BT_CODE_2105.TEST_TEMP[22] := B#16#0;
   S700_1_BT_CODE_2105.TEST_TEMP[23] := B#16#0;
   S700_1_BT_CODE_2105.TEST_TEMP[24] := B#16#0;
   S700_1_BT_CODE_2105.TEST_TEMP[25] := B#16#0;
   S700_1_BT_CODE_2105.TEST_TEMP[26] := B#16#0;
   S700_1_BT_CODE_2105.TEST_TEMP[27] := B#16#0;
   S700_1_BT_CODE_2105.TEST_TEMP[28] := B#16#0;
   S700_1_BT_CODE_2105.TEST_TEMP[29] := B#16#0;
   S700_1_BT_CODE_2105.TEST_TEMP[30] := B#16#0;
   S700_1_BT_CODE_2105.TEST_TEMP[31] := B#16#0;
   S700_1_BT_CODE_2105.TEST_TEMP[32] := B#16#0;
   S700_1_BT_CODE_2105.TEST_TEMP[33] := B#16#0;
   S700_1_BT_CODE_2105.TEST_TEMP[34] := B#16#0;
   S700_1_BT_CODE_2105.TEST_TEMP[35] := B#16#0;
   S700_1_BT_CODE_2105.TEST_TEMP[36] := B#16#0;
   S700_1_BT_CODE_2105.TEST_TEMP[37] := B#16#0;
   S700_1_BT_CODE_2105.TEST_TEMP[38] := B#16#0;
   S700_1_BT_CODE_2105.TEST_TEMP[39] := B#16#0;
   S700_1_BT_CODE_2105.TEST_TEMP[40] := B#16#0;
   S700_1_BT_CODE_2106.STATION_MAIN := W#16#0;
   S700_1_BT_CODE_2106.DISTINCTION_LH_RH := W#16#0;
   S700_1_BT_CODE_2106.STAION_NUMBER := W#16#0;
   S700_1_BT_CODE_2106.BODY_TYPE_1ST := W#16#0;
   S700_1_BT_CODE_2106.BODY_TYPE_OPTION := W#16#0;
   S700_1_BT_CODE_2106.RBT1_STANDARD_WELD_DATA := W#16#0;
   S700_1_BT_CODE_2106.RBT2_STANDARD_WELD_DATA := W#16#0;
   S700_1_BT_CODE_2106.RBT3_STANDARD_WELD_DATA := W#16#0;
   S700_1_BT_CODE_2106.RBT4_STANDARD_WELD_DATA := W#16#0;
   S700_1_BT_CODE_2106.RBT5_STANDARD_WELD_DATA := W#16#0;
   S700_1_BT_CODE_2106.RBT6_STANDARD_WELD_DATA := W#16#0;
   S700_1_BT_CODE_2106.RBT7_STANDARD_WELD_DATA := W#16#0;
   S700_1_BT_CODE_2106.RBT8_STANDARD_WELD_DATA := W#16#0;
   S700_1_BT_CODE_2106.RBT9_STANDARD_WELD_DATA := W#16#0;
   S700_1_BT_CODE_2106.RBT10_STANDARD_WELD_DATA := W#16#0;
   S700_1_BT_CODE_2106.RBT11_STANDARD_WELD_DATA := W#16#0;
   S700_1_BT_CODE_2106.RBT12_STANDARD_WELD_DATA := W#16#0;
   S700_1_BT_CODE_2106.RBT13_STANDARD_WELD_DATA := W#16#0;
   S700_1_BT_CODE_2106.RBT14_STANDARD_WELD_DATA := W#16#0;
   S700_1_BT_CODE_2106.RBT15_STANDARD_WELD_DATA := W#16#0;
   S700_1_BT_CODE_2106.RBT16_STANDARD_WELD_DATA := W#16#0;
   S700_1_BT_CODE_2106.RBT17_STANDARD_WELD_DATA := W#16#0;
   S700_1_BT_CODE_2106.RBT18_STANDARD_WELD_DATA := W#16#0;
   S700_1_BT_CODE_2106.RBT19_STANDARD_WELD_DATA := W#16#0;
   S700_1_BT_CODE_2106.RBT20_STANDARD_WELD_DATA := W#16#0;
   S700_1_BT_CODE_2106.RBT21_STANDARD_WELD_DATA := W#16#0;
   S700_1_BT_CODE_2106.RBT22_STANDARD_WELD_DATA := W#16#0;
   S700_1_BT_CODE_2106.RBT23_STANDARD_WELD_DAT := W#16#0;
   S700_1_BT_CODE_2106.RBT24_STANDARD_WELD_DAT := W#16#0;
   S700_1_BT_CODE_2106.CHK_WORD := W#16#0;
   S700_1_BT_CODE_2106.TEST_TEMP[1] := B#16#0;
   S700_1_BT_CODE_2106.TEST_TEMP[2] := B#16#0;
   S700_1_BT_CODE_2106.TEST_TEMP[3] := B#16#0;
   S700_1_BT_CODE_2106.TEST_TEMP[4] := B#16#0;
   S700_1_BT_CODE_2106.TEST_TEMP[5] := B#16#0;
   S700_1_BT_CODE_2106.TEST_TEMP[6] := B#16#0;
   S700_1_BT_CODE_2106.TEST_TEMP[7] := B#16#0;
   S700_1_BT_CODE_2106.TEST_TEMP[8] := B#16#0;
   S700_1_BT_CODE_2106.TEST_TEMP[9] := B#16#0;
   S700_1_BT_CODE_2106.TEST_TEMP[10] := B#16#0;
   S700_1_BT_CODE_2106.TEST_TEMP[11] := B#16#0;
   S700_1_BT_CODE_2106.TEST_TEMP[12] := B#16#0;
   S700_1_BT_CODE_2106.TEST_TEMP[13] := B#16#0;
   S700_1_BT_CODE_2106.TEST_TEMP[14] := B#16#0;
   S700_1_BT_CODE_2106.TEST_TEMP[15] := B#16#0;
   S700_1_BT_CODE_2106.TEST_TEMP[16] := B#16#0;
   S700_1_BT_CODE_2106.TEST_TEMP[17] := B#16#0;
   S700_1_BT_CODE_2106.TEST_TEMP[18] := B#16#0;
   S700_1_BT_CODE_2106.TEST_TEMP[19] := B#16#0;
   S700_1_BT_CODE_2106.TEST_TEMP[20] := B#16#0;
   S700_1_BT_CODE_2106.TEST_TEMP[21] := B#16#0;
   S700_1_BT_CODE_2106.TEST_TEMP[22] := B#16#0;
   S700_1_BT_CODE_2106.TEST_TEMP[23] := B#16#0;
   S700_1_BT_CODE_2106.TEST_TEMP[24] := B#16#0;
   S700_1_BT_CODE_2106.TEST_TEMP[25] := B#16#0;
   S700_1_BT_CODE_2106.TEST_TEMP[26] := B#16#0;
   S700_1_BT_CODE_2106.TEST_TEMP[27] := B#16#0;
   S700_1_BT_CODE_2106.TEST_TEMP[28] := B#16#0;
   S700_1_BT_CODE_2106.TEST_TEMP[29] := B#16#0;
   S700_1_BT_CODE_2106.TEST_TEMP[30] := B#16#0;
   S700_1_BT_CODE_2106.TEST_TEMP[31] := B#16#0;
   S700_1_BT_CODE_2106.TEST_TEMP[32] := B#16#0;
   S700_1_BT_CODE_2106.TEST_TEMP[33] := B#16#0;
   S700_1_BT_CODE_2106.TEST_TEMP[34] := B#16#0;
   S700_1_BT_CODE_2106.TEST_TEMP[35] := B#16#0;
   S700_1_BT_CODE_2106.TEST_TEMP[36] := B#16#0;
   S700_1_BT_CODE_2106.TEST_TEMP[37] := B#16#0;
   S700_1_BT_CODE_2106.TEST_TEMP[38] := B#16#0;
   S700_1_BT_CODE_2106.TEST_TEMP[39] := B#16#0;
   S700_1_BT_CODE_2106.TEST_TEMP[40] := B#16#0;
   S700_1_BT_CODE_2107.STATION_MAIN := W#16#0;
   S700_1_BT_CODE_2107.DISTINCTION_LH_RH := W#16#0;
   S700_1_BT_CODE_2107.STAION_NUMBER := W#16#0;
   S700_1_BT_CODE_2107.BODY_TYPE_1ST := W#16#0;
   S700_1_BT_CODE_2107.BODY_TYPE_OPTION := W#16#0;
   S700_1_BT_CODE_2107.RBT1_STANDARD_WELD_DATA := W#16#0;
   S700_1_BT_CODE_2107.RBT2_STANDARD_WELD_DATA := W#16#0;
   S700_1_BT_CODE_2107.RBT3_STANDARD_WELD_DATA := W#16#0;
   S700_1_BT_CODE_2107.RBT4_STANDARD_WELD_DATA := W#16#0;
   S700_1_BT_CODE_2107.RBT5_STANDARD_WELD_DATA := W#16#0;
   S700_1_BT_CODE_2107.RBT6_STANDARD_WELD_DATA := W#16#0;
   S700_1_BT_CODE_2107.RBT7_STANDARD_WELD_DATA := W#16#0;
   S700_1_BT_CODE_2107.RBT8_STANDARD_WELD_DATA := W#16#0;
   S700_1_BT_CODE_2107.RBT9_STANDARD_WELD_DATA := W#16#0;
   S700_1_BT_CODE_2107.RBT10_STANDARD_WELD_DATA := W#16#0;
   S700_1_BT_CODE_2107.RBT11_STANDARD_WELD_DATA := W#16#0;
   S700_1_BT_CODE_2107.RBT12_STANDARD_WELD_DATA := W#16#0;
   S700_1_BT_CODE_2107.RBT13_STANDARD_WELD_DATA := W#16#0;
   S700_1_BT_CODE_2107.RBT14_STANDARD_WELD_DATA := W#16#0;
   S700_1_BT_CODE_2107.RBT15_STANDARD_WELD_DATA := W#16#0;
   S700_1_BT_CODE_2107.RBT16_STANDARD_WELD_DATA := W#16#0;
   S700_1_BT_CODE_2107.RBT17_STANDARD_WELD_DATA := W#16#0;
   S700_1_BT_CODE_2107.RBT18_STANDARD_WELD_DATA := W#16#0;
   S700_1_BT_CODE_2107.RBT19_STANDARD_WELD_DATA := W#16#0;
   S700_1_BT_CODE_2107.RBT20_STANDARD_WELD_DATA := W#16#0;
   S700_1_BT_CODE_2107.RBT21_STANDARD_WELD_DATA := W#16#0;
   S700_1_BT_CODE_2107.RBT22_STANDARD_WELD_DATA := W#16#0;
   S700_1_BT_CODE_2107.RBT23_STANDARD_WELD_DAT := W#16#0;
   S700_1_BT_CODE_2107.RBT24_STANDARD_WELD_DAT := W#16#0;
   S700_1_BT_CODE_2107.CHK_WORD := W#16#0;
   S700_1_BT_CODE_2107.TEST_TEMP[1] := B#16#0;
   S700_1_BT_CODE_2107.TEST_TEMP[2] := B#16#0;
   S700_1_BT_CODE_2107.TEST_TEMP[3] := B#16#0;
   S700_1_BT_CODE_2107.TEST_TEMP[4] := B#16#0;
   S700_1_BT_CODE_2107.TEST_TEMP[5] := B#16#0;
   S700_1_BT_CODE_2107.TEST_TEMP[6] := B#16#0;
   S700_1_BT_CODE_2107.TEST_TEMP[7] := B#16#0;
   S700_1_BT_CODE_2107.TEST_TEMP[8] := B#16#0;
   S700_1_BT_CODE_2107.TEST_TEMP[9] := B#16#0;
   S700_1_BT_CODE_2107.TEST_TEMP[10] := B#16#0;
   S700_1_BT_CODE_2107.TEST_TEMP[11] := B#16#0;
   S700_1_BT_CODE_2107.TEST_TEMP[12] := B#16#0;
   S700_1_BT_CODE_2107.TEST_TEMP[13] := B#16#0;
   S700_1_BT_CODE_2107.TEST_TEMP[14] := B#16#0;
   S700_1_BT_CODE_2107.TEST_TEMP[15] := B#16#0;
   S700_1_BT_CODE_2107.TEST_TEMP[16] := B#16#0;
   S700_1_BT_CODE_2107.TEST_TEMP[17] := B#16#0;
   S700_1_BT_CODE_2107.TEST_TEMP[18] := B#16#0;
   S700_1_BT_CODE_2107.TEST_TEMP[19] := B#16#0;
   S700_1_BT_CODE_2107.TEST_TEMP[20] := B#16#0;
   S700_1_BT_CODE_2107.TEST_TEMP[21] := B#16#0;
   S700_1_BT_CODE_2107.TEST_TEMP[22] := B#16#0;
   S700_1_BT_CODE_2107.TEST_TEMP[23] := B#16#0;
   S700_1_BT_CODE_2107.TEST_TEMP[24] := B#16#0;
   S700_1_BT_CODE_2107.TEST_TEMP[25] := B#16#0;
   S700_1_BT_CODE_2107.TEST_TEMP[26] := B#16#0;
   S700_1_BT_CODE_2107.TEST_TEMP[27] := B#16#0;
   S700_1_BT_CODE_2107.TEST_TEMP[28] := B#16#0;
   S700_1_BT_CODE_2107.TEST_TEMP[29] := B#16#0;
   S700_1_BT_CODE_2107.TEST_TEMP[30] := B#16#0;
   S700_1_BT_CODE_2107.TEST_TEMP[31] := B#16#0;
   S700_1_BT_CODE_2107.TEST_TEMP[32] := B#16#0;
   S700_1_BT_CODE_2107.TEST_TEMP[33] := B#16#0;
   S700_1_BT_CODE_2107.TEST_TEMP[34] := B#16#0;
   S700_1_BT_CODE_2107.TEST_TEMP[35] := B#16#0;
   S700_1_BT_CODE_2107.TEST_TEMP[36] := B#16#0;
   S700_1_BT_CODE_2107.TEST_TEMP[37] := B#16#0;
   S700_1_BT_CODE_2107.TEST_TEMP[38] := B#16#0;
   S700_1_BT_CODE_2107.TEST_TEMP[39] := B#16#0;
   S700_1_BT_CODE_2107.TEST_TEMP[40] := B#16#0;
   S700_1_BT_CODE_2108.STATION_MAIN := W#16#0;
   S700_1_BT_CODE_2108.DISTINCTION_LH_RH := W#16#0;
   S700_1_BT_CODE_2108.STAION_NUMBER := W#16#0;
   S700_1_BT_CODE_2108.BODY_TYPE_1ST := W#16#0;
   S700_1_BT_CODE_2108.BODY_TYPE_OPTION := W#16#0;
   S700_1_BT_CODE_2108.RBT1_STANDARD_WELD_DATA := W#16#0;
   S700_1_BT_CODE_2108.RBT2_STANDARD_WELD_DATA := W#16#0;
   S700_1_BT_CODE_2108.RBT3_STANDARD_WELD_DATA := W#16#0;
   S700_1_BT_CODE_2108.RBT4_STANDARD_WELD_DATA := W#16#0;
   S700_1_BT_CODE_2108.RBT5_STANDARD_WELD_DATA := W#16#0;
   S700_1_BT_CODE_2108.RBT6_STANDARD_WELD_DATA := W#16#0;
   S700_1_BT_CODE_2108.RBT7_STANDARD_WELD_DATA := W#16#0;
   S700_1_BT_CODE_2108.RBT8_STANDARD_WELD_DATA := W#16#0;
   S700_1_BT_CODE_2108.RBT9_STANDARD_WELD_DATA := W#16#0;
   S700_1_BT_CODE_2108.RBT10_STANDARD_WELD_DATA := W#16#0;
   S700_1_BT_CODE_2108.RBT11_STANDARD_WELD_DATA := W#16#0;
   S700_1_BT_CODE_2108.RBT12_STANDARD_WELD_DATA := W#16#0;
   S700_1_BT_CODE_2108.RBT13_STANDARD_WELD_DATA := W#16#0;
   S700_1_BT_CODE_2108.RBT14_STANDARD_WELD_DATA := W#16#0;
   S700_1_BT_CODE_2108.RBT15_STANDARD_WELD_DATA := W#16#0;
   S700_1_BT_CODE_2108.RBT16_STANDARD_WELD_DATA := W#16#0;
   S700_1_BT_CODE_2108.RBT17_STANDARD_WELD_DATA := W#16#0;
   S700_1_BT_CODE_2108.RBT18_STANDARD_WELD_DATA := W#16#0;
   S700_1_BT_CODE_2108.RBT19_STANDARD_WELD_DATA := W#16#0;
   S700_1_BT_CODE_2108.RBT20_STANDARD_WELD_DATA := W#16#0;
   S700_1_BT_CODE_2108.RBT21_STANDARD_WELD_DATA := W#16#0;
   S700_1_BT_CODE_2108.RBT22_STANDARD_WELD_DATA := W#16#0;
   S700_1_BT_CODE_2108.RBT23_STANDARD_WELD_DAT := W#16#0;
   S700_1_BT_CODE_2108.RBT24_STANDARD_WELD_DAT := W#16#0;
   S700_1_BT_CODE_2108.CHK_WORD := W#16#0;
   S700_1_BT_CODE_2108.TEST_TEMP[1] := B#16#0;
   S700_1_BT_CODE_2108.TEST_TEMP[2] := B#16#0;
   S700_1_BT_CODE_2108.TEST_TEMP[3] := B#16#0;
   S700_1_BT_CODE_2108.TEST_TEMP[4] := B#16#0;
   S700_1_BT_CODE_2108.TEST_TEMP[5] := B#16#0;
   S700_1_BT_CODE_2108.TEST_TEMP[6] := B#16#0;
   S700_1_BT_CODE_2108.TEST_TEMP[7] := B#16#0;
   S700_1_BT_CODE_2108.TEST_TEMP[8] := B#16#0;
   S700_1_BT_CODE_2108.TEST_TEMP[9] := B#16#0;
   S700_1_BT_CODE_2108.TEST_TEMP[10] := B#16#0;
   S700_1_BT_CODE_2108.TEST_TEMP[11] := B#16#0;
   S700_1_BT_CODE_2108.TEST_TEMP[12] := B#16#0;
   S700_1_BT_CODE_2108.TEST_TEMP[13] := B#16#0;
   S700_1_BT_CODE_2108.TEST_TEMP[14] := B#16#0;
   S700_1_BT_CODE_2108.TEST_TEMP[15] := B#16#0;
   S700_1_BT_CODE_2108.TEST_TEMP[16] := B#16#0;
   S700_1_BT_CODE_2108.TEST_TEMP[17] := B#16#0;
   S700_1_BT_CODE_2108.TEST_TEMP[18] := B#16#0;
   S700_1_BT_CODE_2108.TEST_TEMP[19] := B#16#0;
   S700_1_BT_CODE_2108.TEST_TEMP[20] := B#16#0;
   S700_1_BT_CODE_2108.TEST_TEMP[21] := B#16#0;
   S700_1_BT_CODE_2108.TEST_TEMP[22] := B#16#0;
   S700_1_BT_CODE_2108.TEST_TEMP[23] := B#16#0;
   S700_1_BT_CODE_2108.TEST_TEMP[24] := B#16#0;
   S700_1_BT_CODE_2108.TEST_TEMP[25] := B#16#0;
   S700_1_BT_CODE_2108.TEST_TEMP[26] := B#16#0;
   S700_1_BT_CODE_2108.TEST_TEMP[27] := B#16#0;
   S700_1_BT_CODE_2108.TEST_TEMP[28] := B#16#0;
   S700_1_BT_CODE_2108.TEST_TEMP[29] := B#16#0;
   S700_1_BT_CODE_2108.TEST_TEMP[30] := B#16#0;
   S700_1_BT_CODE_2108.TEST_TEMP[31] := B#16#0;
   S700_1_BT_CODE_2108.TEST_TEMP[32] := B#16#0;
   S700_1_BT_CODE_2108.TEST_TEMP[33] := B#16#0;
   S700_1_BT_CODE_2108.TEST_TEMP[34] := B#16#0;
   S700_1_BT_CODE_2108.TEST_TEMP[35] := B#16#0;
   S700_1_BT_CODE_2108.TEST_TEMP[36] := B#16#0;
   S700_1_BT_CODE_2108.TEST_TEMP[37] := B#16#0;
   S700_1_BT_CODE_2108.TEST_TEMP[38] := B#16#0;
   S700_1_BT_CODE_2108.TEST_TEMP[39] := B#16#0;
   S700_1_BT_CODE_2108.TEST_TEMP[40] := B#16#0;
   S700_1_BT_CODE_2109.STATION_MAIN := W#16#0;
   S700_1_BT_CODE_2109.DISTINCTION_LH_RH := W#16#0;
   S700_1_BT_CODE_2109.STAION_NUMBER := W#16#0;
   S700_1_BT_CODE_2109.BODY_TYPE_1ST := W#16#0;
   S700_1_BT_CODE_2109.BODY_TYPE_OPTION := W#16#0;
   S700_1_BT_CODE_2109.RBT1_STANDARD_WELD_DATA := W#16#0;
   S700_1_BT_CODE_2109.RBT2_STANDARD_WELD_DATA := W#16#0;
   S700_1_BT_CODE_2109.RBT3_STANDARD_WELD_DATA := W#16#0;
   S700_1_BT_CODE_2109.RBT4_STANDARD_WELD_DATA := W#16#0;
   S700_1_BT_CODE_2109.RBT5_STANDARD_WELD_DATA := W#16#0;
   S700_1_BT_CODE_2109.RBT6_STANDARD_WELD_DATA := W#16#0;
   S700_1_BT_CODE_2109.RBT7_STANDARD_WELD_DATA := W#16#0;
   S700_1_BT_CODE_2109.RBT8_STANDARD_WELD_DATA := W#16#0;
   S700_1_BT_CODE_2109.RBT9_STANDARD_WELD_DATA := W#16#0;
   S700_1_BT_CODE_2109.RBT10_STANDARD_WELD_DATA := W#16#0;
   S700_1_BT_CODE_2109.RBT11_STANDARD_WELD_DATA := W#16#0;
   S700_1_BT_CODE_2109.RBT12_STANDARD_WELD_DATA := W#16#0;
   S700_1_BT_CODE_2109.RBT13_STANDARD_WELD_DATA := W#16#0;
   S700_1_BT_CODE_2109.RBT14_STANDARD_WELD_DATA := W#16#0;
   S700_1_BT_CODE_2109.RBT15_STANDARD_WELD_DATA := W#16#0;
   S700_1_BT_CODE_2109.RBT16_STANDARD_WELD_DATA := W#16#0;
   S700_1_BT_CODE_2109.RBT17_STANDARD_WELD_DATA := W#16#0;
   S700_1_BT_CODE_2109.RBT18_STANDARD_WELD_DATA := W#16#0;
   S700_1_BT_CODE_2109.RBT19_STANDARD_WELD_DATA := W#16#0;
   S700_1_BT_CODE_2109.RBT20_STANDARD_WELD_DATA := W#16#0;
   S700_1_BT_CODE_2109.RBT21_STANDARD_WELD_DATA := W#16#0;
   S700_1_BT_CODE_2109.RBT22_STANDARD_WELD_DATA := W#16#0;
   S700_1_BT_CODE_2109.RBT23_STANDARD_WELD_DAT := W#16#0;
   S700_1_BT_CODE_2109.RBT24_STANDARD_WELD_DAT := W#16#0;
   S700_1_BT_CODE_2109.CHK_WORD := W#16#0;
   S700_1_BT_CODE_2109.TEST_TEMP[1] := B#16#0;
   S700_1_BT_CODE_2109.TEST_TEMP[2] := B#16#0;
   S700_1_BT_CODE_2109.TEST_TEMP[3] := B#16#0;
   S700_1_BT_CODE_2109.TEST_TEMP[4] := B#16#0;
   S700_1_BT_CODE_2109.TEST_TEMP[5] := B#16#0;
   S700_1_BT_CODE_2109.TEST_TEMP[6] := B#16#0;
   S700_1_BT_CODE_2109.TEST_TEMP[7] := B#16#0;
   S700_1_BT_CODE_2109.TEST_TEMP[8] := B#16#0;
   S700_1_BT_CODE_2109.TEST_TEMP[9] := B#16#0;
   S700_1_BT_CODE_2109.TEST_TEMP[10] := B#16#0;
   S700_1_BT_CODE_2109.TEST_TEMP[11] := B#16#0;
   S700_1_BT_CODE_2109.TEST_TEMP[12] := B#16#0;
   S700_1_BT_CODE_2109.TEST_TEMP[13] := B#16#0;
   S700_1_BT_CODE_2109.TEST_TEMP[14] := B#16#0;
   S700_1_BT_CODE_2109.TEST_TEMP[15] := B#16#0;
   S700_1_BT_CODE_2109.TEST_TEMP[16] := B#16#0;
   S700_1_BT_CODE_2109.TEST_TEMP[17] := B#16#0;
   S700_1_BT_CODE_2109.TEST_TEMP[18] := B#16#0;
   S700_1_BT_CODE_2109.TEST_TEMP[19] := B#16#0;
   S700_1_BT_CODE_2109.TEST_TEMP[20] := B#16#0;
   S700_1_BT_CODE_2109.TEST_TEMP[21] := B#16#0;
   S700_1_BT_CODE_2109.TEST_TEMP[22] := B#16#0;
   S700_1_BT_CODE_2109.TEST_TEMP[23] := B#16#0;
   S700_1_BT_CODE_2109.TEST_TEMP[24] := B#16#0;
   S700_1_BT_CODE_2109.TEST_TEMP[25] := B#16#0;
   S700_1_BT_CODE_2109.TEST_TEMP[26] := B#16#0;
   S700_1_BT_CODE_2109.TEST_TEMP[27] := B#16#0;
   S700_1_BT_CODE_2109.TEST_TEMP[28] := B#16#0;
   S700_1_BT_CODE_2109.TEST_TEMP[29] := B#16#0;
   S700_1_BT_CODE_2109.TEST_TEMP[30] := B#16#0;
   S700_1_BT_CODE_2109.TEST_TEMP[31] := B#16#0;
   S700_1_BT_CODE_2109.TEST_TEMP[32] := B#16#0;
   S700_1_BT_CODE_2109.TEST_TEMP[33] := B#16#0;
   S700_1_BT_CODE_2109.TEST_TEMP[34] := B#16#0;
   S700_1_BT_CODE_2109.TEST_TEMP[35] := B#16#0;
   S700_1_BT_CODE_2109.TEST_TEMP[36] := B#16#0;
   S700_1_BT_CODE_2109.TEST_TEMP[37] := B#16#0;
   S700_1_BT_CODE_2109.TEST_TEMP[38] := B#16#0;
   S700_1_BT_CODE_2109.TEST_TEMP[39] := B#16#0;
